LIN {X 0,Y 301.473,Z 710.898,A -85,B 0,C 180,E1 14594.697,E2 14594.697} C_VEL
LIN {X 0,Y 299.686,Z 720.643,A -85,B 0,C 180,E1 14592.72,E2 14592.72} C_VEL
LIN {X 0,Y 297.823,Z 729.269,A -85,B 0,C 180,E1 14590.444,E2 14590.444} C_VEL
LIN {X 0,Y 296.157,Z 735.724,A -85,B 0,C 180,E1 14588.151,E2 14588.151} C_VEL
LIN {X 0,Y 294.632,Z 740.781,A -85,B 0,C 180,E1 14585.647,E2 14585.647} C_VEL
LIN {X 0,Y 293.317,Z 744.193,A -85,B 0,C 180,E1 14582.93,E2 14582.93} C_VEL
LIN {X 0,Y 292.262,Z 745.687,A -85,B 0,C 180,E1 14579.999,E2 14579.999} C_VEL
LIN {X 0,Y 291.583,Z 745.107,A -85,B 0,C 180,E1 14577.168,E2 14577.168} C_VEL
LIN {X 0,Y 291.215,Z 742.755,A -85,B 0,C 180,E1 14574.483,E2 14574.483} C_VEL
LIN {X 0,Y 291.115,Z 738.842,A -85,B 0,C 180,E1 14571.904,E2 14571.904} C_VEL
LIN {X 0,Y 291.269,Z 732.598,A -85,B 0,C 180,E1 14569.116,E2 14569.116} C_VEL
LIN {X 0,Y 291.687,Z 724.621,A -85,B 0,C 180,E1 14566.52,E2 14566.52} C_VEL
LIN {X 0,Y 292.312,Z 714.997,A -85,B 0,C 180,E1 14564.118,E2 14564.118} C_VEL
LIN {X 0,Y 293.088,Z 703.694,A -85,B 0,C 180,E1 14561.913,E2 14561.913} C_VEL
LIN {X 0,Y 293.954,Z 690.528,A -85,B 0,C 180,E1 14559.906,E2 14559.906} C_VEL
LIN {X 0,Y 294.781,Z 675.92,A -85,B 0,C 180,E1 14558.197,E2 14558.197} C_VEL
LIN {X 0,Y 295.446,Z 660.979,A -85,B 0,C 180,E1 14556.885,E2 14556.885} C_VEL
LIN {X 0,Y 295.895,Z 644.769,A -85,B 0,C 180,E1 14555.878,E2 14555.878} C_VEL
LIN {X 0,Y 296.067,Z 626.386,A -85,B 0,C 180,E1 14555.173,E2 14555.173} C_VEL
LIN {X 0,Y 297.336,Z 577.945,A -85,B 0,C 180,E1 14553.621,E2 14553.621} C_VEL
LIN {X 0,Y 298.083,Z 578.111,A -85,B 0,C 180,E1 14553.289,E2 14553.289} C_VEL
LIN {X 0,Y 299.719,Z 576.086,A -85,B 0,C 180,E1 14552.857,E2 14552.857} C_VEL
LIN {X 0,Y 302.62,Z 570.153,A -85,B 0,C 180,E1 14552.375,E2 14552.375} C_VEL
LIN {X 0,Y 306.801,Z 558.743,A -85,B 0,C 180,E1 14551.96,E2 14551.96} C_VEL
LIN {X 0,Y 307.694,Z 556.167,A -85,B 0,C 180,E1 14551.888,E2 14551.888} C_VEL
LIN {X 0,Y 310.325,Z 552.374,A -85,B 0,C 180,E1 14551.283,E2 14551.283} C_VEL
LIN {X 0,Y 313.629,Z 545.368,A -85,B 0,C 180,E1 14550.753,E2 14550.753} C_VEL
LIN {X 0,Y 317.925,Z 533.318,A -85,B 0,C 180,E1 14550.308,E2 14550.308} C_VEL
LIN {X 0,Y 319.018,Z 529.98,A -85,B 0,C 180,E1 14550.213,E2 14550.213} C_VEL
LIN {X 0,Y 323.323,Z 523.899,A -85,B 0,C 180,E1 14549.272,E2 14549.272} C_VEL
LIN {X 0,Y 329.072,Z 514.334,A -85,B 0,C 180,E1 14548.185,E2 14548.185} C_VEL
LIN {X 0,Y 333.692,Z 509.138,A -85,B 0,C 180,E1 14547.182,E2 14547.182} C_VEL
LIN {X 0,Y 338.897,Z 501.157,A -85,B 0,C 180,E1 14546.236,E2 14546.236} C_VEL
LIN {X 0,Y 340.375,Z 498.972,A -85,B 0,C 180,E1 14545.971,E2 14545.971} C_VEL
LIN {X 0,Y 345.61,Z 492.984,A -85,B 0,C 180,E1 14544.958,E2 14544.958} C_VEL
LIN {X 0,Y 351.852,Z 483.792,A -85,B 0,C 180,E1 14543.917,E2 14543.917} C_VEL
LIN {X 0,Y 356.859,Z 478.438,A -85,B 0,C 180,E1 14543.023,E2 14543.023} C_VEL
LIN {X 0,Y 350.683,Z 533.515,A -85,B 0,C 180,E1 14541.496,E2 14541.496} C_VEL
LIN {X 0,Y 343.595,Z 587.069,A -85,B 0,C 180,E1 14539.73,E2 14539.73} C_VEL
LIN {X 0,Y 340.274,Z 612.573,A -85,B 0,C 180,E1 14538.644,E2 14538.644} C_VEL
LIN {X 0,Y 336.94,Z 632.228,A -85,B 0,C 180,E1 14537.512,E2 14537.512} C_VEL
LIN {X 0,Y 332.931,Z 651.111,A -85,B 0,C 180,E1 14536.119,E2 14536.119} C_VEL
LIN {X 0,Y 328.102,Z 670.254,A -85,B 0,C 180,E1 14534.334,E2 14534.334} C_VEL
LIN {X 0,Y 322.92,Z 688.102,A -85,B 0,C 180,E1 14532.266,E2 14532.266} C_VEL
LIN {X 0,Y 317.65,Z 704.404,A -85,B 0,C 180,E1 14529.951,E2 14529.951} C_VEL
LIN {X 0,Y 312.389,Z 719.507,A -85,B 0,C 180,E1 14527.339,E2 14527.339} C_VEL
LIN {X 0,Y 307.364,Z 733.168,A -85,B 0,C 180,E1 14524.474,E2 14524.474} C_VEL
LIN {X 0,Y 302.603,Z 745.779,A -85,B 0,C 180,E1 14521.249,E2 14521.249} C_VEL
LIN {X 0,Y 298.41,Z 756.887,A -85,B 0,C 180,E1 14517.758,E2 14517.758} C_VEL
LIN {X 0,Y 294.914,Z 766.473,A -85,B 0,C 180,E1 14514.007,E2 14514.007} C_VEL
LIN {X 0,Y 292.324,Z 774.116,A -85,B 0,C 180,E1 14510.21,E2 14510.21} C_VEL
LIN {X 0,Y 290.465,Z 780.308,A -85,B 0,C 180,E1 14506.176,E2 14506.176} C_VEL
LIN {X 0,Y 289.38,Z 784.674,A -85,B 0,C 180,E1 14502.167,E2 14502.167} C_VEL
LIN {X 0,Y 288.847,Z 787.269,A -85,B 0,C 180,E1 14498.36,E2 14498.36} C_VEL
LIN {X 0,Y 288.632,Z 788.437,A -85,B 0,C 180,E1 14494.371,E2 14494.371} C_VEL
LIN {X 0,Y 288.641,Z 788.017,A -85,B 0,C 180,E1 14490.397,E2 14490.397} C_VEL
LIN {X 0,Y 288.874,Z 786.163,A -85,B 0,C 180,E1 14486.627,E2 14486.627} C_VEL
LIN {X 0,Y 289.451,Z 782.871,A -85,B 0,C 180,E1 14482.856,E2 14482.856} C_VEL
LIN {X 0,Y 290.598,Z 777.745,A -85,B 0,C 180,E1 14478.891,E2 14478.891} C_VEL
LIN {X 0,Y 291.846,Z 772.956,A -85,B 0,C 180,E1 14476.075,E2 14476.075} C_VEL
LIN {X 0,Y 291.661,Z 770.405,A -85,B 0,C 180,E1 14474.638,E2 14474.638} C_VEL
LIN {X 0,Y 288.214,Z 763.219,A -85,B 0,C 180,E1 14470.745,E2 14470.745} C_VEL
LIN {X 0,Y 288.512,Z 760.327,A -85,B 0,C 180,E1 14469.546,E2 14469.546} C_VEL
LIN {X 0,Y 292.227,Z 749.899,A -85,B 0,C 180,E1 14465.973,E2 14465.973} C_VEL
LIN {X 0,Y 296.474,Z 738.2,A -85,B 0,C 180,E1 14462.699,E2 14462.699} C_VEL
LIN {X 0,Y 301.185,Z 725.063,A -85,B 0,C 180,E1 14459.672,E2 14459.672} C_VEL
LIN {X 0,Y 306.278,Z 710.292,A -85,B 0,C 180,E1 14456.871,E2 14456.871} C_VEL
LIN {X 0,Y 311.276,Z 694.805,A -85,B 0,C 180,E1 14454.451,E2 14454.451} C_VEL
LIN {X 0,Y 316.243,Z 677.951,A -85,B 0,C 180,E1 14452.281,E2 14452.281} C_VEL
LIN {X 0,Y 320.912,Z 660.2,A -85,B 0,C 180,E1 14450.42,E2 14450.42} C_VEL
LIN {X 0,Y 324.977,Z 642.253,A -85,B 0,C 180,E1 14448.897,E2 14448.897} C_VEL
LIN {X 0,Y 328.596,Z 622.858,A -85,B 0,C 180,E1 14447.59,E2 14447.59} C_VEL
LIN {X 0,Y 331.499,Z 602.817,A -85,B 0,C 180,E1 14446.562,E2 14446.562} C_VEL
LIN {X 0,Y 336.631,Z 562.875,A -85,B 0,C 180,E1 14445.046,E2 14445.046} C_VEL
LIN {X 0,Y 343.508,Z 506.974,A -85,B 0,C 180,E1 14443.314,E2 14443.314} C_VEL
LIN {X 0,Y 348.719,Z 454.242,A -85,B 0,C 180,E1 14441.938,E2 14441.938} C_VEL
LIN {X 0,Y 352.555,Z 400.926,A -85,B 0,C 180,E1 14440.775,E2 14440.775} C_VEL
LIN {X 0,Y 352.938,Z 393.306,A -85,B 0,C 180,E1 14440.603,E2 14440.603} C_VEL
LIN {X 0,Y 344.835,Z 382.448,A -85,B 0,C 180,E1 14438.327,E2 14438.327} C_VEL
LIN {X 0,Y 335.306,Z 391.656,A -85,B 0,C 180,E1 14436.188,E2 14436.188} C_VEL
LIN {X 0,Y 329.497,Z 398.011,A -85,B 0,C 180,E1 14434.785,E2 14434.785} C_VEL
LIN {X 0,Y 325.165,Z 402.639,A -85,B 0,C 180,E1 14433.66,E2 14433.66} C_VEL
LIN {X 0,Y 319.752,Z 409.849,A -85,B 0,C 180,E1 14432.219,E2 14432.219} C_VEL
LIN {X 0,Y 314.779,Z 421.202,A -85,B 0,C 180,E1 14431.023,E2 14431.023} C_VEL
LIN {X 0,Y 311.088,Z 427.898,A -85,B 0,C 180,E1 14429.987,E2 14429.987} C_VEL
LIN {X 0,Y 308.623,Z 431.225,A -85,B 0,C 180,E1 14429.196,E2 14429.196} C_VEL
LIN {X 0,Y 303.63,Z 444,A -85,B 0,C 180,E1 14427.853,E2 14427.853} C_VEL
LIN {X 0,Y 300.278,Z 450.967,A -85,B 0,C 180,E1 14426.794,E2 14426.794} C_VEL
LIN {X 0,Y 298.518,Z 453.454,A -85,B 0,C 180,E1 14426.133,E2 14426.133} C_VEL
LIN {X 0,Y 297.997,Z 453.855,A -85,B 0,C 180,E1 14425.888,E2 14425.888} C_VEL
LIN {X 0,Y 296.772,Z 468.599,A -85,B 0,C 180,E1 14424.405,E2 14424.405} C_VEL
LIN {X 0,Y 296.008,Z 473.564,A -85,B 0,C 180,E1 14424.006,E2 14424.006} C_VEL
LIN {X 0,Y 290.441,Z 604.08,A -85,B 0,C 180,E1 14419.652,E2 14419.652} C_VEL
LIN {X 0,Y 290.011,Z 625.296,A -85,B 0,C 180,E1 14418.793,E2 14418.793} C_VEL
LIN {X 0,Y 289.326,Z 642.963,A -85,B 0,C 180,E1 14417.706,E2 14417.706} C_VEL
LIN {X 0,Y 288.352,Z 660.558,A -85,B 0,C 180,E1 14416.209,E2 14416.209} C_VEL
LIN {X 0,Y 287.212,Z 677.45,A -85,B 0,C 180,E1 14414.311,E2 14414.311} C_VEL
LIN {X 0,Y 286.035,Z 692.745,A -85,B 0,C 180,E1 14412.108,E2 14412.108} C_VEL
LIN {X 0,Y 284.951,Z 706.521,A -85,B 0,C 180,E1 14409.598,E2 14409.598} C_VEL
LIN {X 0,Y 284.135,Z 717.555,A -85,B 0,C 180,E1 14407.075,E2 14407.075} C_VEL
LIN {X 0,Y 283.579,Z 726.784,A -85,B 0,C 180,E1 14404.45,E2 14404.45} C_VEL
LIN {X 0,Y 283.252,Z 735.102,A -85,B 0,C 180,E1 14401.417,E2 14401.417} C_VEL
LIN {X 0,Y 283.252,Z 741.235,A -85,B 0,C 180,E1 14398.383,E2 14398.383} C_VEL
LIN {X 0,Y 283.544,Z 745.254,A -85,B 0,C 180,E1 14395.551,E2 14395.551} C_VEL
LIN {X 0,Y 284.166,Z 747.725,A -85,B 0,C 180,E1 14392.52,E2 14392.52} C_VEL
LIN {X 0,Y 285.075,Z 748.436,A -85,B 0,C 180,E1 14389.696,E2 14389.696} C_VEL
LIN {X 0,Y 286.424,Z 747.35,A -85,B 0,C 180,E1 14386.68,E2 14386.68} C_VEL
LIN {X 0,Y 288.052,Z 744.664,A -85,B 0,C 180,E1 14383.878,E2 14383.878} C_VEL
LIN {X 0,Y 290.06,Z 740.16,A -85,B 0,C 180,E1 14381.094,E2 14381.094} C_VEL
LIN {X 0,Y 292.467,Z 733.68,A -85,B 0,C 180,E1 14378.333,E2 14378.333} C_VEL
LIN {X 0,Y 295.04,Z 725.576,A -85,B 0,C 180,E1 14375.792,E2 14375.792} C_VEL
LIN {X 0,Y 297.684,Z 715.934,A -85,B 0,C 180,E1 14373.467,E2 14373.467} C_VEL
LIN {X 0,Y 300.337,Z 704.849,A -85,B 0,C 180,E1 14371.355,E2 14371.355} C_VEL
LIN {X 0,Y 303.037,Z 691.567,A -85,B 0,C 180,E1 14369.352,E2 14369.352} C_VEL
LIN {X 0,Y 305.593,Z 676.279,A -85,B 0,C 180,E1 14367.549,E2 14367.549} C_VEL
LIN {X 0,Y 307.814,Z 659.516,A -85,B 0,C 180,E1 14366.035,E2 14366.035} C_VEL
LIN {X 0,Y 309.452,Z 643.901,A -85,B 0,C 180,E1 14364.949,E2 14364.949} C_VEL
LIN {X 0,Y 312.209,Z 641.947,A -85,B 0,C 180,E1 14364.574,E2 14364.574} C_VEL
LIN {X 0,Y 315.963,Z 637.407,A -85,B 0,C 180,E1 14364.279,E2 14364.279} C_VEL
LIN {X 0,Y 318.626,Z 632.886,A -85,B 0,C 180,E1 14364.181,E2 14364.181} C_VEL
LIN {X 0,Y 322.084,Z 629.461,A -85,B 0,C 180,E1 14363.817,E2 14363.817} C_VEL
LIN {X 0,Y 326.321,Z 623.421,A -85,B 0,C 180,E1 14363.529,E2 14363.529} C_VEL
LIN {X 0,Y 329.749,Z 617.515,A -85,B 0,C 180,E1 14363.375,E2 14363.375} C_VEL
LIN {X 0,Y 334.495,Z 611.357,A -85,B 0,C 180,E1 14362.965,E2 14362.965} C_VEL
LIN {X 0,Y 339.904,Z 601.538,A -85,B 0,C 180,E1 14362.673,E2 14362.673} C_VEL
LIN {X 0,Y 341.058,Z 599.168,A -85,B 0,C 180,E1 14362.623,E2 14362.623} C_VEL
LIN {X 0,Y 336.007,Z 627.852,A -85,B 0,C 180,E1 14361.432,E2 14361.432} C_VEL
LIN {X 0,Y 330.753,Z 653.868,A -85,B 0,C 180,E1 14360.025,E2 14360.025} C_VEL
LIN {X 0,Y 325.14,Z 679.325,A -85,B 0,C 180,E1 14358.27,E2 14358.27} C_VEL
LIN {X 0,Y 319.358,Z 703.464,A -85,B 0,C 180,E1 14356.219,E2 14356.219} C_VEL
LIN {X 0,Y 314.203,Z 722.714,A -85,B 0,C 180,E1 14354.179,E2 14354.179} C_VEL
LIN {X 0,Y 309.087,Z 739.953,A -85,B 0,C 180,E1 14351.926,E2 14351.926} C_VEL
LIN {X 0,Y 303.589,Z 756.816,A -85,B 0,C 180,E1 14349.224,E2 14349.224} C_VEL
LIN {X 0,Y 298.58,Z 771.612,A -85,B 0,C 180,E1 14346.351,E2 14346.351} C_VEL
LIN {X 0,Y 293.647,Z 785.695,A -85,B 0,C 180,E1 14343.011,E2 14343.011} C_VEL
LIN {X 0,Y 289.342,Z 798.276,A -85,B 0,C 180,E1 14339.387,E2 14339.387} C_VEL
LIN {X 0,Y 285.795,Z 809.244,A -85,B 0,C 180,E1 14335.488,E2 14335.488} C_VEL
LIN {X 0,Y 283.125,Z 818.695,A -85,B 0,C 180,E1 14331.33,E2 14331.33} C_VEL
LIN {X 0,Y 281.424,Z 826.219,A -85,B 0,C 180,E1 14327.117,E2 14327.117} C_VEL
LIN {X 0,Y 280.547,Z 832.143,A -85,B 0,C 180,E1 14322.766,E2 14322.766} C_VEL
LIN {X 0,Y 280.318,Z 836.176,A -85,B 0,C 180,E1 14318.616,E2 14318.616} C_VEL
LIN {X 0,Y 280.394,Z 838.536,A -85,B 0,C 180,E1 14314.704,E2 14314.704} C_VEL
LIN {X 0,Y 280.478,Z 839.547,A -85,B 0,C 180,E1 14310.817,E2 14310.817} C_VEL
LIN {X 0,Y 280.429,Z 839.233,A -85,B 0,C 180,E1 14306.934,E2 14306.934} C_VEL
LIN {X 0,Y 280.319,Z 837.595,A -85,B 0,C 180,E1 14303.034,E2 14303.034} C_VEL
LIN {X 0,Y 280.377,Z 834.425,A -85,B 0,C 180,E1 14298.897,E2 14298.897} C_VEL
LIN {X 0,Y 280.979,Z 829.386,A -85,B 0,C 180,E1 14294.521,E2 14294.521} C_VEL
LIN {X 0,Y 282.433,Z 822.567,A -85,B 0,C 180,E1 14290.132,E2 14290.132} C_VEL
LIN {X 0,Y 284.789,Z 814.229,A -85,B 0,C 180,E1 14285.967,E2 14285.967} C_VEL
LIN {X 0,Y 288.424,Z 803.331,A -85,B 0,C 180,E1 14281.645,E2 14281.645} C_VEL
LIN {X 0,Y 292.672,Z 791.63,A -85,B 0,C 180,E1 14277.912,E2 14277.912} C_VEL
LIN {X 0,Y 297.922,Z 777.604,A -85,B 0,C 180,E1 14274.27,E2 14274.27} C_VEL
LIN {X 0,Y 303.283,Z 763.18,A -85,B 0,C 180,E1 14271.215,E2 14271.215} C_VEL
LIN {X 0,Y 309.187,Z 746.554,A -85,B 0,C 180,E1 14268.332,E2 14268.332} C_VEL
LIN {X 0,Y 314.815,Z 729.546,A -85,B 0,C 180,E1 14265.928,E2 14265.928} C_VEL
LIN {X 0,Y 320.081,Z 711.951,A -85,B 0,C 180,E1 14263.905,E2 14263.905} C_VEL
LIN {X 0,Y 324.783,Z 694.187,A -85,B 0,C 180,E1 14262.235,E2 14262.235} C_VEL
LIN {X 0,Y 330.423,Z 671.409,A -85,B 0,C 180,E1 14260.444,E2 14260.444} C_VEL
LIN {X 0,Y 336.265,Z 645.855,A -85,B 0,C 180,E1 14258.827,E2 14258.827} C_VEL
LIN {X 0,Y 341.881,Z 618.451,A -85,B 0,C 180,E1 14257.485,E2 14257.485} C_VEL
LIN {X 0,Y 346.787,Z 589.883,A -85,B 0,C 180,E1 14256.411,E2 14256.411} C_VEL
LIN {X 0,Y 349.983,Z 567.917,A -85,B 0,C 180,E1 14255.797,E2 14255.797} C_VEL
LIN {X 0,Y 353.901,Z 543.241,A -85,B 0,C 180,E1 14255.513,E2 14255.513} C_VEL
LIN {X 0,Y 355.166,Z 534.693,A -85,B 0,C 180,E1 14255.47,E2 14255.47} C_VEL
LIN {X 0,Y 346.998,Z 514.246,A -85,B 0,C 180,E1 14252.898,E2 14252.898} C_VEL
LIN {X 0,Y 342.19,Z 498.864,A -85,B 0,C 180,E1 14251.115,E2 14251.115} C_VEL
LIN {X 0,Y 338.758,Z 503.075,A -85,B 0,C 180,E1 14250.361,E2 14250.361} C_VEL
LIN {X 0,Y 333.41,Z 513.045,A -85,B 0,C 180,E1 14249.262,E2 14249.262} C_VEL
LIN {X 0,Y 331.124,Z 516.93,A -85,B 0,C 180,E1 14248.754,E2 14248.754} C_VEL
LIN {X 0,Y 325.481,Z 529.287,A -85,B 0,C 180,E1 14247.611,E2 14247.611} C_VEL
LIN {X 0,Y 318.157,Z 545.033,A -85,B 0,C 180,E1 14246.189,E2 14246.189} C_VEL
LIN {X 0,Y 311.572,Z 565.14,A -85,B 0,C 180,E1 14245.506,E2 14245.506} C_VEL
LIN {X 0,Y 307.707,Z 574.04,A -85,B 0,C 180,E1 14244.962,E2 14244.962} C_VEL
LIN {X 0,Y 306.249,Z 576.987,A -85,B 0,C 180,E1 14244.676,E2 14244.676} C_VEL
LIN {X 0,Y 301.442,Z 633.673,A -85,B 0,C 180,E1 14242.435,E2 14242.435} C_VEL
LIN {X 0,Y 300.381,Z 660.053,A -85,B 0,C 180,E1 14241.196,E2 14241.196} C_VEL
LIN {X 0,Y 299.511,Z 674.161,A -85,B 0,C 180,E1 14240.213,E2 14240.213} C_VEL
LIN {X 0,Y 298.152,Z 688.209,A -85,B 0,C 180,E1 14238.881,E2 14238.881} C_VEL
LIN {X 0,Y 296.484,Z 701.18,A -85,B 0,C 180,E1 14237.263,E2 14237.263} C_VEL
LIN {X 0,Y 294.653,Z 712.217,A -85,B 0,C 180,E1 14235.481,E2 14235.481} C_VEL
LIN {X 0,Y 292.688,Z 722.167,A -85,B 0,C 180,E1 14233.432,E2 14233.432} C_VEL
LIN {X 0,Y 290.642,Z 730.739,A -85,B 0,C 180,E1 14231.107,E2 14231.107} C_VEL
LIN {X 0,Y 288.692,Z 737.689,A -85,B 0,C 180,E1 14228.564,E2 14228.564} C_VEL
LIN {X 0,Y 287.034,Z 742.578,A -85,B 0,C 180,E1 14225.998,E2 14225.998} C_VEL
LIN {X 0,Y 285.603,Z 745.838,A -85,B 0,C 180,E1 14223.21,E2 14223.21} C_VEL
LIN {X 0,Y 284.522,Z 747.18,A -85,B 0,C 180,E1 14220.402,E2 14220.402} C_VEL
LIN {X 0,Y 283.767,Z 746.63,A -85,B 0,C 180,E1 14217.576,E2 14217.576} C_VEL
LIN {X 0,Y 283.351,Z 744.475,A -85,B 0,C 180,E1 14214.938,E2 14214.938} C_VEL
LIN {X 0,Y 283.185,Z 740.308,A -85,B 0,C 180,E1 14212.084,E2 14212.084} C_VEL
LIN {X 0,Y 283.317,Z 734.044,A -85,B 0,C 180,E1 14209.219,E2 14209.219} C_VEL
LIN {X 0,Y 283.727,Z 726.067,A -85,B 0,C 180,E1 14206.55,E2 14206.55} C_VEL
LIN {X 0,Y 284.358,Z 716.452,A -85,B 0,C 180,E1 14204.081,E2 14204.081} C_VEL
LIN {X 0,Y 285.149,Z 705.131,A -85,B 0,C 180,E1 14201.815,E2 14201.815} C_VEL
LIN {X 0,Y 286.038,Z 691.955,A -85,B 0,C 180,E1 14199.753,E2 14199.753} C_VEL
LIN {X 0,Y 286.902,Z 677.151,A -85,B 0,C 180,E1 14197.976,E2 14197.976} C_VEL
LIN {X 0,Y 287.597,Z 661.945,A -85,B 0,C 180,E1 14196.611,E2 14196.611} C_VEL
LIN {X 0,Y 288.063,Z 645.959,A -85,B 0,C 180,E1 14195.595,E2 14195.595} C_VEL
LIN {X 0,Y 288.255,Z 627.249,A -85,B 0,C 180,E1 14194.854,E2 14194.854} C_VEL
LIN {X 0,Y 288.75,Z 603.42,A -85,B 0,C 180,E1 14194.021,E2 14194.021} C_VEL
LIN {X 0,Y 289.539,Z 603.619,A -85,B 0,C 180,E1 14193.656,E2 14193.656} C_VEL
LIN {X 0,Y 291.248,Z 601.636,A -85,B 0,C 180,E1 14193.201,E2 14193.201} C_VEL
LIN {X 0,Y 294.153,Z 596.042,A -85,B 0,C 180,E1 14192.725,E2 14192.725} C_VEL
LIN {X 0,Y 298.315,Z 585.446,A -85,B 0,C 180,E1 14192.34,E2 14192.34} C_VEL
LIN {X 0,Y 298.798,Z 584.326,A -85,B 0,C 180,E1 14192.28,E2 14192.28} C_VEL
LIN {X 0,Y 301.447,Z 580.726,A -85,B 0,C 180,E1 14191.658,E2 14191.658} C_VEL
LIN {X 0,Y 304.858,Z 574.047,A -85,B 0,C 180,E1 14191.116,E2 14191.116} C_VEL
LIN {X 0,Y 309.255,Z 562.611,A -85,B 0,C 180,E1 14190.682,E2 14190.682} C_VEL
LIN {X 0,Y 310.163,Z 560.384,A -85,B 0,C 180,E1 14190.579,E2 14190.579} C_VEL
LIN {X 0,Y 313.547,Z 554.777,A -85,B 0,C 180,E1 14189.93,E2 14189.93} C_VEL
LIN {X 0,Y 317.447,Z 546.013,A -85,B 0,C 180,E1 14189.398,E2 14189.398} C_VEL
LIN {X 0,Y 321.678,Z 534.312,A -85,B 0,C 180,E1 14188.989,E2 14188.989} C_VEL
LIN {X 0,Y 327.825,Z 525.172,A -85,B 0,C 180,E1 14187.792,E2 14187.792} C_VEL
LIN {X 0,Y 330.859,Z 520.239,A -85,B 0,C 180,E1 14187.252,E2 14187.252} C_VEL
LIN {X 0,Y 336.05,Z 514.248,A -85,B 0,C 180,E1 14186.193,E2 14186.193} C_VEL
LIN {X 0,Y 341.775,Z 505.555,A -85,B 0,C 180,E1 14185.216,E2 14185.216} C_VEL
LIN {X 0,Y 348.007,Z 498.402,A -85,B 0,C 180,E1 14184.067,E2 14184.067} C_VEL
LIN {X 0,Y 350.504,Z 495.083,A -85,B 0,C 180,E1 14183.652,E2 14183.652} C_VEL
LIN {X 0,Y 343.831,Z 549.112,A -85,B 0,C 180,E1 14182.074,E2 14182.074} C_VEL
LIN {X 0,Y 337.573,Z 594.457,A -85,B 0,C 180,E1 14180.488,E2 14180.488} C_VEL
LIN {X 0,Y 334.298,Z 617.469,A -85,B 0,C 180,E1 14179.438,E2 14179.438} C_VEL
LIN {X 0,Y 330.58,Z 637.491,A -85,B 0,C 180,E1 14178.207,E2 14178.207} C_VEL
LIN {X 0,Y 326.131,Z 656.786,A -85,B 0,C 180,E1 14176.685,E2 14176.685} C_VEL
LIN {X 0,Y 321.332,Z 674.476,A -85,B 0,C 180,E1 14174.938,E2 14174.938} C_VEL
LIN {X 0,Y 316.045,Z 691.625,A -85,B 0,C 180,E1 14172.859,E2 14172.859} C_VEL
LIN {X 0,Y 310.315,Z 708.386,A -85,B 0,C 180,E1 14170.364,E2 14170.364} C_VEL
LIN {X 0,Y 304.734,Z 723.436,A -85,B 0,C 180,E1 14167.61,E2 14167.61} C_VEL
LIN {X 0,Y 299.447,Z 736.974,A -85,B 0,C 180,E1 14164.586,E2 14164.586} C_VEL
LIN {X 0,Y 294.434,Z 749.487,A -85,B 0,C 180,E1 14161.155,E2 14161.155} C_VEL
LIN {X 0,Y 290.14,Z 760.241,A -85,B 0,C 180,E1 14157.502,E2 14157.502} C_VEL
LIN {X 0,Y 286.662,Z 769.297,A -85,B 0,C 180,E1 14153.648,E2 14153.648} C_VEL
LIN {X 0,Y 284.112,Z 776.483,A -85,B 0,C 180,E1 14149.746,E2 14149.746} C_VEL
LIN {X 0,Y 282.318,Z 782.213,A -85,B 0,C 180,E1 14145.615,E2 14145.615} C_VEL
LIN {X 0,Y 281.299,Z 786.19,A -85,B 0,C 180,E1 14141.481,E2 14141.481} C_VEL
LIN {X 0,Y 280.83,Z 788.452,A -85,B 0,C 180,E1 14137.57,E2 14137.57} C_VEL
LIN {X 0,Y 280.655,Z 789.247,A -85,B 0,C 180,E1 14133.472,E2 14133.472} C_VEL
LIN {X 0,Y 280.715,Z 788.494,A -85,B 0,C 180,E1 14129.592,E2 14129.592} C_VEL
LIN {X 0,Y 281.014,Z 786.329,A -85,B 0,C 180,E1 14125.715,E2 14125.715} C_VEL
LIN {X 0,Y 281.775,Z 782.486,A -85,B 0,C 180,E1 14121.635,E2 14121.635} C_VEL
LIN {X 0,Y 283.171,Z 776.95,A -85,B 0,C 180,E1 14117.562,E2 14117.562} C_VEL
LIN {X 0,Y 285.395,Z 769.595,A -85,B 0,C 180,E1 14113.514,E2 14113.514} C_VEL
LIN {X 0,Y 288.361,Z 760.758,A -85,B 0,C 180,E1 14109.712,E2 14109.712} C_VEL
LIN {X 0,Y 288.512,Z 760.327,A -85,B 0,C 180,E1 14109.546,E2 14109.546} C_VEL
LIN {X 0,Y 288.845,Z 756.908,A -85,B 0,C 180,E1 14108.166,E2 14108.166} C_VEL
LIN {X 0,Y 286.851,Z 748.129,A -85,B 0,C 180,E1 14104.586,E2 14104.586} C_VEL
LIN {X 0,Y 287.58,Z 743.998,A -85,B 0,C 180,E1 14103.272,E2 14103.272} C_VEL
LIN {X 0,Y 292.4,Z 731.332,A -85,B 0,C 180,E1 14100.05,E2 14100.05} C_VEL
LIN {X 0,Y 297.715,Z 716.915,A -85,B 0,C 180,E1 14097.039,E2 14097.039} C_VEL
LIN {X 0,Y 303.299,Z 700.848,A -85,B 0,C 180,E1 14094.303,E2 14094.303} C_VEL
LIN {X 0,Y 308.555,Z 684.249,A -85,B 0,C 180,E1 14091.998,E2 14091.998} C_VEL
LIN {X 0,Y 313.53,Z 666.737,A -85,B 0,C 180,E1 14090.014,E2 14090.014} C_VEL
LIN {X 0,Y 318.143,Z 647.977,A -85,B 0,C 180,E1 14088.302,E2 14088.302} C_VEL
LIN {X 0,Y 322.06,Z 628.877,A -85,B 0,C 180,E1 14086.921,E2 14086.921} C_VEL
LIN {X 0,Y 325.211,Z 609.441,A -85,B 0,C 180,E1 14085.832,E2 14085.832} C_VEL
LIN {X 0,Y 329.868,Z 574.362,A -85,B 0,C 180,E1 14084.399,E2 14084.399} C_VEL
LIN {X 0,Y 337.033,Z 520.261,A -85,B 0,C 180,E1 14082.638,E2 14082.638} C_VEL
LIN {X 0,Y 342.733,Z 467.47,A -85,B 0,C 180,E1 14081.194,E2 14081.194} C_VEL
LIN {X 0,Y 346.898,Z 416.197,A -85,B 0,C 180,E1 14080.026,E2 14080.026} C_VEL
LIN {X 0,Y 348.024,Z 397.545,A -85,B 0,C 180,E1 14079.629,E2 14079.629} C_VEL
LIN {X 0,Y 343.595,Z 391.743,A -85,B 0,C 180,E1 14078.358,E2 14078.358} C_VEL
LIN {X 0,Y 336.308,Z 399.076,A -85,B 0,C 180,E1 14076.751,E2 14076.751} C_VEL
LIN {X 0,Y 330.857,Z 404.904,A -85,B 0,C 180,E1 14075.467,E2 14075.467} C_VEL
LIN {X 0,Y 325.093,Z 411.229,A -85,B 0,C 180,E1 14074.014,E2 14074.014} C_VEL
LIN {X 0,Y 321.814,Z 415.767,A -85,B 0,C 180,E1 14073.177,E2 14073.177} C_VEL
LIN {X 0,Y 316.612,Z 427.101,A -85,B 0,C 180,E1 14071.963,E2 14071.963} C_VEL
LIN {X 0,Y 312.483,Z 434.231,A -85,B 0,C 180,E1 14070.848,E2 14070.848} C_VEL
LIN {X 0,Y 310.32,Z 437.349,A -85,B 0,C 180,E1 14070.202,E2 14070.202} C_VEL
LIN {X 0,Y 305.021,Z 450.105,A -85,B 0,C 180,E1 14068.835,E2 14068.835} C_VEL
LIN {X 0,Y 301.378,Z 457.188,A -85,B 0,C 180,E1 14067.73,E2 14067.73} C_VEL
LIN {X 0,Y 299.019,Z 460.764,A -85,B 0,C 180,E1 14066.902,E2 14066.902} C_VEL
LIN {X 0,Y 293.641,Z 475.605,A -85,B 0,C 180,E1 14065.448,E2 14065.448} C_VEL
LIN {X 0,Y 290.016,Z 488.364,A -85,B 0,C 180,E1 14064.711,E2 14064.711} C_VEL
LIN {X 0,Y 288.155,Z 493.193,A -85,B 0,C 180,E1 14064.171,E2 14064.171} C_VEL
LIN {X 0,Y 287.441,Z 494.48,A -85,B 0,C 180,E1 14063.86,E2 14063.86} C_VEL
LIN {X 0,Y 282.665,Z 604.848,A -85,B 0,C 180,E1 14060.014,E2 14060.014} C_VEL
LIN {X 0,Y 282.2,Z 626.495,A -85,B 0,C 180,E1 14059.112,E2 14059.112} C_VEL
LIN {X 0,Y 281.492,Z 644.075,A -85,B 0,C 180,E1 14058.001,E2 14058.001} C_VEL
LIN {X 0,Y 280.503,Z 661.451,A -85,B 0,C 180,E1 14056.491,E2 14056.491} C_VEL
LIN {X 0,Y 279.367,Z 677.882,A -85,B 0,C 180,E1 14054.616,E2 14054.616} C_VEL
LIN {X 0,Y 278.247,Z 692.07,A -85,B 0,C 180,E1 14052.557,E2 14052.557} C_VEL
LIN {X 0,Y 277.222,Z 704.752,A -85,B 0,C 180,E1 14050.285,E2 14050.285} C_VEL
LIN {X 0,Y 276.333,Z 716.457,A -85,B 0,C 180,E1 14047.695,E2 14047.695} C_VEL
LIN {X 0,Y 275.671,Z 726.876,A -85,B 0,C 180,E1 14044.786,E2 14044.786} C_VEL
LIN {X 0,Y 275.331,Z 735.054,A -85,B 0,C 180,E1 14041.874,E2 14041.874} C_VEL
LIN {X 0,Y 275.303,Z 741.687,A -85,B 0,C 180,E1 14038.752,E2 14038.752} C_VEL
LIN {X 0,Y 275.65,Z 746.567,A -85,B 0,C 180,E1 14035.424,E2 14035.424} C_VEL
LIN {X 0,Y 276.337,Z 749.212,A -85,B 0,C 180,E1 14032.307,E2 14032.307} C_VEL
LIN {X 0,Y 277.424,Z 750.081,A -85,B 0,C 180,E1 14029.199,E2 14029.199} C_VEL
LIN {X 0,Y 278.922,Z 749.03,A -85,B 0,C 180,E1 14026.104,E2 14026.104} C_VEL
LIN {X 0,Y 280.733,Z 746.415,A -85,B 0,C 180,E1 14023.233,E2 14023.233} C_VEL
LIN {X 0,Y 283.122,Z 741.563,A -85,B 0,C 180,E1 14020.183,E2 14020.183} C_VEL
LIN {X 0,Y 285.606,Z 735.511,A -85,B 0,C 180,E1 14017.552,E2 14017.552} C_VEL
LIN {X 0,Y 288.404,Z 727.547,A -85,B 0,C 180,E1 14014.979,E2 14014.979} C_VEL
LIN {X 0,Y 291.297,Z 718.064,A -85,B 0,C 180,E1 14012.617,E2 14012.617} C_VEL
LIN {X 0,Y 294.244,Z 707.059,A -85,B 0,C 180,E1 14010.448,E2 14010.448} C_VEL
LIN {X 0,Y 297.309,Z 693.608,A -85,B 0,C 180,E1 14008.357,E2 14008.357} C_VEL
LIN {X 0,Y 300.13,Z 678.694,A -85,B 0,C 180,E1 14006.541,E2 14006.541} C_VEL
LIN {X 0,Y 302.578,Z 662.738,A -85,B 0,C 180,E1 14005.036,E2 14005.036} C_VEL
LIN {X 0,Y 303.267,Z 657.999,A -85,B 0,C 180,E1 14004.647,E2 14004.647} C_VEL
LIN {X 0,Y 306.275,Z 656.194,A -85,B 0,C 180,E1 14004.243,E2 14004.243} C_VEL
LIN {X 0,Y 309.957,Z 652.257,A -85,B 0,C 180,E1 14003.935,E2 14003.935} C_VEL
LIN {X 0,Y 312.119,Z 649.255,A -85,B 0,C 180,E1 14003.831,E2 14003.831} C_VEL
LIN {X 0,Y 316.297,Z 645.47,A -85,B 0,C 180,E1 14003.411,E2 14003.411} C_VEL
LIN {X 0,Y 320.875,Z 639.296,A -85,B 0,C 180,E1 14003.142,E2 14003.142} C_VEL
LIN {X 0,Y 322.154,Z 637.336,A -85,B 0,C 180,E1 14003.091,E2 14003.091} C_VEL
LIN {X 0,Y 326.855,Z 632.084,A -85,B 0,C 180,E1 14002.689,E2 14002.689} C_VEL
LIN {X 0,Y 330.624,Z 626.5,A -85,B 0,C 180,E1 14002.481,E2 14002.481} C_VEL
LIN {X 0,Y 325.202,Z 652.699,A -85,B 0,C 180,E1 14001.066,E2 14001.066} C_VEL
LIN {X 0,Y 319.17,Z 679.283,A -85,B 0,C 180,E1 13999.229,E2 13999.229} C_VEL
LIN {X 0,Y 313.157,Z 703.459,A -85,B 0,C 180,E1 13997.151,E2 13997.151} C_VEL
LIN {X 0,Y 307.796,Z 722.673,A -85,B 0,C 180,E1 13995.086,E2 13995.086} C_VEL
LIN {X 0,Y 302.427,Z 739.918,A -85,B 0,C 180,E1 13992.782,E2 13992.782} C_VEL
LIN {X 0,Y 296.751,Z 756.625,A -85,B 0,C 180,E1 13990.057,E2 13990.057} C_VEL
LIN {X 0,Y 291.514,Z 771.316,A -85,B 0,C 180,E1 13987.133,E2 13987.133} C_VEL
LIN {X 0,Y 286.357,Z 785.361,A -85,B 0,C 180,E1 13983.723,E2 13983.723} C_VEL
LIN {X 0,Y 281.843,Z 797.896,A -85,B 0,C 180,E1 13980.014,E2 13980.014} C_VEL
LIN {X 0,Y 277.943,Z 809.34,A -85,B 0,C 180,E1 13975.803,E2 13975.803} C_VEL
LIN {X 0,Y 275.183,Z 818.64,A -85,B 0,C 180,E1 13971.529,E2 13971.529} C_VEL
LIN {X 0,Y 273.382,Z 826.298,A -85,B 0,C 180,E1 13967.013,E2 13967.013} C_VEL
LIN {X 0,Y 272.538,Z 831.954,A -85,B 0,C 180,E1 13962.614,E2 13962.614} C_VEL
LIN {X 0,Y 272.343,Z 835.86,A -85,B 0,C 180,E1 13958.232,E2 13958.232} C_VEL
LIN {X 0,Y 272.436,Z 838.043,A -85,B 0,C 180,E1 13954.209,E2 13954.209} C_VEL
LIN {X 0,Y 272.515,Z 838.872,A -85,B 0,C 180,E1 13950.21,E2 13950.21} C_VEL
LIN {X 0,Y 272.432,Z 838.365,A -85,B 0,C 180,E1 13946.212,E2 13946.212} C_VEL
LIN {X 0,Y 272.323,Z 836.525,A -85,B 0,C 180,E1 13942.192,E2 13942.192} C_VEL
LIN {X 0,Y 272.46,Z 833.082,A -85,B 0,C 180,E1 13937.926,E2 13937.926} C_VEL
LIN {X 0,Y 273.25,Z 827.791,A -85,B 0,C 180,E1 13933.416,E2 13933.416} C_VEL
LIN {X 0,Y 274.972,Z 820.697,A -85,B 0,C 180,E1 13928.9,E2 13928.9} C_VEL
LIN {X 0,Y 277.841,Z 811.555,A -85,B 0,C 180,E1 13924.415,E2 13924.415} C_VEL
LIN {X 0,Y 281.531,Z 801.392,A -85,B 0,C 180,E1 13920.418,E2 13920.418} C_VEL
LIN {X 0,Y 286.3,Z 789.042,A -85,B 0,C 180,E1 13916.51,E2 13916.51} C_VEL
LIN {X 0,Y 291.689,Z 775.475,A -85,B 0,C 180,E1 13913.004,E2 13913.004} C_VEL
LIN {X 0,Y 297.361,Z 760.789,A -85,B 0,C 180,E1 13909.916,E2 13909.916} C_VEL
LIN {X 0,Y 303.32,Z 744.747,A -85,B 0,C 180,E1 13907.147,E2 13907.147} C_VEL
LIN {X 0,Y 309.117,Z 727.872,A -85,B 0,C 180,E1 13904.766,E2 13904.766} C_VEL
LIN {X 0,Y 314.8,Z 709.501,A -85,B 0,C 180,E1 13902.668,E2 13902.668} C_VEL
LIN {X 0,Y 320.058,Z 690.177,A -85,B 0,C 180,E1 13900.886,E2 13900.886} C_VEL
LIN {X 0,Y 326.231,Z 665.644,A -85,B 0,C 180,E1 13899.036,E2 13899.036} C_VEL
LIN {X 0,Y 332.388,Z 638.845,A -85,B 0,C 180,E1 13897.425,E2 13897.425} C_VEL
LIN {X 0,Y 338.137,Z 610.893,A -85,B 0,C 180,E1 13896.147,E2 13896.147} C_VEL
LIN {X 0,Y 343.219,Z 580.059,A -85,B 0,C 180,E1 13895.054,E2 13895.054} C_VEL
LIN {X 0,Y 346.437,Z 559.693,A -85,B 0,C 180,E1 13894.617,E2 13894.617} C_VEL
LIN {X 0,Y 349.938,Z 537.417,A -85,B 0,C 180,E1 13894.428,E2 13894.428} C_VEL
LIN {X 0,Y 342.577,Z 517.901,A -85,B 0,C 180,E1 13891.937,E2 13891.937} C_VEL
LIN {X 0,Y 340.204,Z 510.75,A -85,B 0,C 180,E1 13891.05,E2 13891.05} C_VEL
LIN {X 0,Y 334.85,Z 520.05,A -85,B 0,C 180,E1 13889.96,E2 13889.96} C_VEL
LIN {X 0,Y 333.264,Z 523.16,A -85,B 0,C 180,E1 13889.647,E2 13889.647} C_VEL
LIN {X 0,Y 327.358,Z 535.331,A -85,B 0,C 180,E1 13888.505,E2 13888.505} C_VEL
LIN {X 0,Y 320.768,Z 549.42,A -85,B 0,C 180,E1 13887.33,E2 13887.33} C_VEL
LIN {X 0,Y 315.352,Z 566.098,A -85,B 0,C 180,E1 13886.834,E2 13886.834} C_VEL
LIN {X 0,Y 310.723,Z 576.895,A -85,B 0,C 180,E1 13886.26,E2 13886.26} C_VEL
LIN {X 0,Y 308.716,Z 580.825,A -85,B 0,C 180,E1 13885.964,E2 13885.964} C_VEL
LIN {X 0,Y 303.588,Z 593.844,A -85,B 0,C 180,E1 13885.546,E2 13885.546} C_VEL
LIN {X 0,Y 299.711,Z 601.292,A -85,B 0,C 180,E1 13885.04,E2 13885.04} C_VEL
LIN {X 0,Y 298.254,Z 603.855,A -85,B 0,C 180,E1 13884.76,E2 13884.76} C_VEL
LIN {X 0,Y 295.067,Z 643.386,A -85,B 0,C 180,E1 13883.073,E2 13883.073} C_VEL
LIN {X 0,Y 294.154,Z 663.595,A -85,B 0,C 180,E1 13882.021,E2 13882.021} C_VEL
LIN {X 0,Y 293.007,Z 678.517,A -85,B 0,C 180,E1 13880.891,E2 13880.891} C_VEL
LIN {X 0,Y 291.519,Z 691.847,A -85,B 0,C 180,E1 13879.536,E2 13879.536} C_VEL
LIN {X 0,Y 289.673,Z 704.196,A -85,B 0,C 180,E1 13877.89,E2 13877.89} C_VEL
LIN {X 0,Y 287.667,Z 715.108,A -85,B 0,C 180,E1 13876.04,E2 13876.04} C_VEL
LIN {X 0,Y 285.566,Z 724.576,A -85,B 0,C 180,E1 13873.98,E2 13873.98} C_VEL
LIN {X 0,Y 283.369,Z 732.965,A -85,B 0,C 180,E1 13871.602,E2 13871.602} C_VEL
LIN {X 0,Y 281.254,Z 739.698,A -85,B 0,C 180,E1 13868.998,E2 13868.998} C_VEL
LIN {X 0,Y 279.457,Z 744.41,A -85,B 0,C 180,E1 13866.367,E2 13866.367} C_VEL
LIN {X 0,Y 278.003,Z 747.37,A -85,B 0,C 180,E1 13863.711,E2 13863.711} C_VEL
LIN {X 0,Y 276.797,Z 748.677,A -85,B 0,C 180,E1 13860.827,E2 13860.827} C_VEL
LIN {X 0,Y 275.949,Z 748.116,A -85,B 0,C 180,E1 13857.923,E2 13857.923} C_VEL
LIN {X 0,Y 275.467,Z 745.943,A -85,B 0,C 180,E1 13855.21,E2 13855.21} C_VEL
LIN {X 0,Y 275.257,Z 741.764,A -85,B 0,C 180,E1 13852.275,E2 13852.275} C_VEL
LIN {X 0,Y 275.363,Z 735.475,A -85,B 0,C 180,E1 13849.327,E2 13849.327} C_VEL
LIN {X 0,Y 275.76,Z 727.453,A -85,B 0,C 180,E1 13846.581,E2 13846.581} C_VEL
LIN {X 0,Y 276.395,Z 717.789,A -85,B 0,C 180,E1 13844.041,E2 13844.041} C_VEL
LIN {X 0,Y 277.204,Z 706.462,A -85,B 0,C 180,E1 13841.711,E2 13841.711} C_VEL
LIN {X 0,Y 278.12,Z 693.297,A -85,B 0,C 180,E1 13839.59,E2 13839.59} C_VEL
LIN {X 0,Y 279.009,Z 678.64,A -85,B 0,C 180,E1 13837.773,E2 13837.773} C_VEL
LIN {X 0,Y 279.743,Z 663.222,A -85,B 0,C 180,E1 13836.346,E2 13836.346} C_VEL
LIN {X 0,Y 280.237,Z 647.18,A -85,B 0,C 180,E1 13835.298,E2 13835.298} C_VEL
LIN {X 0,Y 280.442,Z 628.642,A -85,B 0,C 180,E1 13834.539,E2 13834.539} C_VEL
LIN {X 0,Y 280.505,Z 625.823,A -85,B 0,C 180,E1 13834.413,E2 13834.413} C_VEL
LIN {X 0,Y 281.175,Z 626.12,A -85,B 0,C 180,E1 13834.062,E2 13834.062} C_VEL
LIN {X 0,Y 282.257,Z 625.31,A -85,B 0,C 180,E1 13833.717,E2 13833.717} C_VEL
LIN {X 0,Y 284.459,Z 622.113,A -85,B 0,C 180,E1 13833.261,E2 13833.261} C_VEL
LIN {X 0,Y 288.017,Z 614.601,A -85,B 0,C 180,E1 13832.823,E2 13832.823} C_VEL
LIN {X 0,Y 289.967,Z 609.958,A -85,B 0,C 180,E1 13832.646,E2 13832.646} C_VEL
LIN {X 0,Y 292.732,Z 606.496,A -85,B 0,C 180,E1 13831.988,E2 13831.988} C_VEL
LIN {X 0,Y 296.156,Z 600.209,A -85,B 0,C 180,E1 13831.44,E2 13831.44} C_VEL
LIN {X 0,Y 300.532,Z 589.625,A -85,B 0,C 180,E1 13831.023,E2 13831.023} C_VEL
LIN {X 0,Y 301.986,Z 587.429,A -85,B 0,C 180,E1 13830.739,E2 13830.739} C_VEL
LIN {X 0,Y 305.598,Z 581.32,A -85,B 0,C 180,E1 13830.101,E2 13830.101} C_VEL
LIN {X 0,Y 309.787,Z 571.921,A -85,B 0,C 180,E1 13829.601,E2 13829.601} C_VEL
LIN {X 0,Y 312.658,Z 564.488,A -85,B 0,C 180,E1 13829.345,E2 13829.345} C_VEL
LIN {X 0,Y 316.675,Z 557.525,A -85,B 0,C 180,E1 13828.655,E2 13828.655} C_VEL
LIN {X 0,Y 321.061,Z 547.578,A -85,B 0,C 180,E1 13828.125,E2 13828.125} C_VEL
LIN {X 0,Y 324.452,Z 538.542,A -85,B 0,C 180,E1 13827.808,E2 13827.808} C_VEL
LIN {X 0,Y 332.113,Z 526.868,A -85,B 0,C 180,E1 13826.438,E2 13826.438} C_VEL
LIN {X 0,Y 338.866,Z 518.862,A -85,B 0,C 180,E1 13825.158,E2 13825.158} C_VEL
LIN {X 0,Y 344.103,Z 511.177,A -85,B 0,C 180,E1 13824.299,E2 13824.299} C_VEL
LIN {X 0,Y 337.008,Z 563.704,A -85,B 0,C 180,E1 13822.685,E2 13822.685} C_VEL
LIN {X 0,Y 331.401,Z 602.831,A -85,B 0,C 180,E1 13821.219,E2 13821.219} C_VEL
LIN {X 0,Y 328.109,Z 623.797,A -85,B 0,C 180,E1 13820.169,E2 13820.169} C_VEL
LIN {X 0,Y 324.022,Z 643.673,A -85,B 0,C 180,E1 13818.845,E2 13818.845} C_VEL
LIN {X 0,Y 319.293,Z 662.469,A -85,B 0,C 180,E1 13817.253,E2 13817.253} C_VEL
LIN {X 0,Y 314.005,Z 680.415,A -85,B 0,C 180,E1 13815.357,E2 13815.357} C_VEL
LIN {X 0,Y 308.215,Z 697.802,A -85,B 0,C 180,E1 13813.082,E2 13813.082} C_VEL
LIN {X 0,Y 302.173,Z 714.23,A -85,B 0,C 180,E1 13810.432,E2 13810.432} C_VEL
LIN {X 0,Y 296.439,Z 728.711,A -85,B 0,C 180,E1 13807.567,E2 13807.567} C_VEL
LIN {X 0,Y 290.89,Z 742.107,A -85,B 0,C 180,E1 13804.313,E2 13804.313} C_VEL
LIN {X 0,Y 285.811,Z 754.101,A -85,B 0,C 180,E1 13800.715,E2 13800.715} C_VEL
LIN {X 0,Y 281.459,Z 764.497,A -85,B 0,C 180,E1 13796.818,E2 13796.818} C_VEL
LIN {X 0,Y 277.952,Z 773.226,A -85,B 0,C 180,E1 13792.638,E2 13792.638} C_VEL
LIN {X 0,Y 275.483,Z 779.974,A -85,B 0,C 180,E1 13788.407,E2 13788.407} C_VEL
LIN {X 0,Y 273.937,Z 784.912,A -85,B 0,C 180,E1 13784.155,E2 13784.155} C_VEL
LIN {X 0,Y 273.103,Z 788.151,A -85,B 0,C 180,E1 13779.908,E2 13779.908} C_VEL
LIN {X 0,Y 272.747,Z 789.76,A -85,B 0,C 180,E1 13775.681,E2 13775.681} C_VEL
LIN {X 0,Y 272.683,Z 789.78,A -85,B 0,C 180,E1 13771.681,E2 13771.681} C_VEL
LIN {X 0,Y 272.855,Z 788.386,A -85,B 0,C 180,E1 13767.69,E2 13767.69} C_VEL
LIN {X 0,Y 273.404,Z 785.385,A -85,B 0,C 180,E1 13763.49,E2 13763.49} C_VEL
LIN {X 0,Y 274.528,Z 780.737,A -85,B 0,C 180,E1 13759.295,E2 13759.295} C_VEL
LIN {X 0,Y 276.443,Z 774.337,A -85,B 0,C 180,E1 13755.12,E2 13755.12} C_VEL
LIN {X 0,Y 279.272,Z 766.05,A -85,B 0,C 180,E1 13750.986,E2 13750.986} C_VEL
LIN {X 0,Y 282.898,Z 756.229,A -85,B 0,C 180,E1 13747.121,E2 13747.121} C_VEL
LIN {X 0,Y 287.217,Z 744.92,A -85,B 0,C 180,E1 13743.539,E2 13743.539} C_VEL
LIN {X 0,Y 287.58,Z 743.998,A -85,B 0,C 180,E1 13743.272,E2 13743.272} C_VEL
LIN {X 0,Y 288.419,Z 739.809,A -85,B 0,C 180,E1 13741.981,E2 13741.981} C_VEL
LIN {X 0,Y 287.689,Z 729.061,A -85,B 0,C 180,E1 13738.597,E2 13738.597} C_VEL
LIN {X 0,Y 288.738,Z 724.137,A -85,B 0,C 180,E1 13737.423,E2 13737.423} C_VEL
LIN {X 0,Y 294.204,Z 709.55,A -85,B 0,C 180,E1 13734.653,E2 13734.653} C_VEL
LIN {X 0,Y 299.789,Z 693.424,A -85,B 0,C 180,E1 13732.144,E2 13732.144} C_VEL
LIN {X 0,Y 305.024,Z 676.761,A -85,B 0,C 180,E1 13730.023,E2 13730.023} C_VEL
LIN {X 0,Y 309.98,Z 658.858,A -85,B 0,C 180,E1 13728.169,E2 13728.169} C_VEL
LIN {X 0,Y 314.406,Z 640.091,A -85,B 0,C 180,E1 13726.613,E2 13726.613} C_VEL
LIN {X 0,Y 318.071,Z 620.993,A -85,B 0,C 180,E1 13725.366,E2 13725.366} C_VEL
LIN {X 0,Y 321.191,Z 600.053,A -85,B 0,C 180,E1 13724.332,E2 13724.332} C_VEL
LIN {X 0,Y 327.19,Z 557.637,A -85,B 0,C 180,E1 13722.728,E2 13722.728} C_VEL
LIN {X 0,Y 334.079,Z 504.443,A -85,B 0,C 180,E1 13721.084,E2 13721.084} C_VEL
LIN {X 0,Y 339.378,Z 453.367,A -85,B 0,C 180,E1 13719.757,E2 13719.757} C_VEL
LIN {X 0,Y 343.234,Z 401.981,A -85,B 0,C 180,E1 13718.64,E2 13718.64} C_VEL
LIN {X 0,Y 342.54,Z 401.308,A -85,B 0,C 180,E1 13718.444,E2 13718.444} C_VEL
LIN {X 0,Y 337.955,Z 405.766,A -85,B 0,C 180,E1 13717.445,E2 13717.445} C_VEL
LIN {X 0,Y 331.963,Z 412.122,A -85,B 0,C 180,E1 13716.075,E2 13716.075} C_VEL
LIN {X 0,Y 326.679,Z 417.792,A -85,B 0,C 180,E1 13714.781,E2 13714.781} C_VEL
LIN {X 0,Y 323.967,Z 421.633,A -85,B 0,C 180,E1 13714.121,E2 13714.121} C_VEL
LIN {X 0,Y 318.501,Z 432.976,A -85,B 0,C 180,E1 13712.895,E2 13712.895} C_VEL
LIN {X 0,Y 314.067,Z 440.364,A -85,B 0,C 180,E1 13711.742,E2 13711.742} C_VEL
LIN {X 0,Y 312.205,Z 443.126,A -85,B 0,C 180,E1 13711.223,E2 13711.223} C_VEL
LIN {X 0,Y 306.576,Z 455.955,A -85,B 0,C 180,E1 13709.837,E2 13709.837} C_VEL
LIN {X 0,Y 302.508,Z 463.394,A -85,B 0,C 180,E1 13708.665,E2 13708.665} C_VEL
LIN {X 0,Y 300.417,Z 466.675,A -85,B 0,C 180,E1 13707.989,E2 13707.989} C_VEL
LIN {X 0,Y 295.796,Z 478.856,A -85,B 0,C 180,E1 13706.819,E2 13706.819} C_VEL
LIN {X 0,Y 291.949,Z 491.785,A -85,B 0,C 180,E1 13706.083,E2 13706.083} C_VEL
LIN {X 0,Y 289.552,Z 497.904,A -85,B 0,C 180,E1 13705.436,E2 13705.436} C_VEL
LIN {X 0,Y 288.94,Z 499.487,A -85,B 0,C 180,E1 13705.267,E2 13705.267} C_VEL
LIN {X 0,Y 284.219,Z 517.151,A -85,B 0,C 180,E1 13704.652,E2 13704.652} C_VEL
LIN {X 0,Y 280.712,Z 527.957,A -85,B 0,C 180,E1 13703.972,E2 13703.972} C_VEL
LIN {X 0,Y 278.683,Z 532.72,A -85,B 0,C 180,E1 13703.385,E2 13703.385} C_VEL
LIN {X 0,Y 277.855,Z 534.032,A -85,B 0,C 180,E1 13702.997,E2 13702.997} C_VEL
LIN {X 0,Y 274.849,Z 608.06,A -85,B 0,C 180,E1 13700.302,E2 13700.302} C_VEL
LIN {X 0,Y 274.384,Z 627.955,A -85,B 0,C 180,E1 13699.429,E2 13699.429} C_VEL
LIN {X 0,Y 273.622,Z 645.744,A -85,B 0,C 180,E1 13698.256,E2 13698.256} C_VEL
LIN {X 0,Y 272.614,Z 662.671,A -85,B 0,C 180,E1 13696.734,E2 13696.734} C_VEL
LIN {X 0,Y 271.394,Z 679.681,A -85,B 0,C 180,E1 13694.727,E2 13694.727} C_VEL
LIN {X 0,Y 270.154,Z 695.104,A -85,B 0,C 180,E1 13692.397,E2 13692.397} C_VEL
LIN {X 0,Y 269.055,Z 708.518,A -85,B 0,C 180,E1 13689.844,E2 13689.844} C_VEL
LIN {X 0,Y 268.237,Z 719.387,A -85,B 0,C 180,E1 13687.282,E2 13687.282} C_VEL
LIN {X 0,Y 267.663,Z 728.912,A -85,B 0,C 180,E1 13684.5,E2 13684.5} C_VEL
LIN {X 0,Y 267.354,Z 736.955,A -85,B 0,C 180,E1 13681.501,E2 13681.501} C_VEL
LIN {X 0,Y 267.378,Z 743.164,A -85,B 0,C 180,E1 13678.501,E2 13678.501} C_VEL
LIN {X 0,Y 267.795,Z 748.11,A -85,B 0,C 180,E1 13675.074,E2 13675.074} C_VEL
LIN {X 0,Y 268.576,Z 750.807,A -85,B 0,C 180,E1 13671.868,E2 13671.868} C_VEL
LIN {X 0,Y 269.796,Z 751.735,A -85,B 0,C 180,E1 13668.673,E2 13668.673} C_VEL
LIN {X 0,Y 271.463,Z 750.76,A -85,B 0,C 180,E1 13665.496,E2 13665.496} C_VEL
LIN {X 0,Y 273.624,Z 747.941,A -85,B 0,C 180,E1 13662.345,E2 13662.345} C_VEL
LIN {X 0,Y 276.296,Z 743.053,A -85,B 0,C 180,E1 13659.229,E2 13659.229} C_VEL
LIN {X 0,Y 279.064,Z 736.88,A -85,B 0,C 180,E1 13656.524,E2 13656.524} C_VEL
LIN {X 0,Y 282.141,Z 729.01,A -85,B 0,C 180,E1 13653.933,E2 13653.933} C_VEL
LIN {X 0,Y 285.612,Z 718.681,A -85,B 0,C 180,E1 13651.341,E2 13651.341} C_VEL
LIN {X 0,Y 289.118,Z 706.546,A -85,B 0,C 180,E1 13648.984,E2 13648.984} C_VEL
LIN {X 0,Y 292.411,Z 693.227,A -85,B 0,C 180,E1 13646.95,E2 13646.95} C_VEL
LIN {X 0,Y 295.397,Z 679.004,A -85,B 0,C 180,E1 13645.227,E2 13645.227} C_VEL
LIN {X 0,Y 297.023,Z 670.818,A -85,B 0,C 180,E1 13644.384,E2 13644.384} C_VEL
LIN {X 0,Y 300.481,Z 668.743,A -85,B 0,C 180,E1 13643.917,E2 13643.917} C_VEL
LIN {X 0,Y 304.305,Z 665.028,A -85,B 0,C 180,E1 13643.611,E2 13643.611} C_VEL
LIN {X 0,Y 305.826,Z 663.462,A -85,B 0,C 180,E1 13643.486,E2 13643.486} C_VEL
LIN {X 0,Y 310.382,Z 659.696,A -85,B 0,C 180,E1 13643.026,E2 13643.026} C_VEL
LIN {X 0,Y 315.512,Z 653.756,A -85,B 0,C 180,E1 13642.695,E2 13642.695} C_VEL
LIN {X 0,Y 320.358,Z 648.952,A -85,B 0,C 180,E1 13642.302,E2 13642.302} C_VEL
LIN {X 0,Y 314.181,Z 675.435,A -85,B 0,C 180,E1 13640.511,E2 13640.511} C_VEL
LIN {X 0,Y 308.221,Z 699.129,A -85,B 0,C 180,E1 13638.535,E2 13638.535} C_VEL
LIN {X 0,Y 302.87,Z 718,A -85,B 0,C 180,E1 13636.576,E2 13636.576} C_VEL
LIN {X 0,Y 297.182,Z 735.946,A -85,B 0,C 180,E1 13634.264,E2 13634.264} C_VEL
LIN {X 0,Y 291.233,Z 752.979,A -85,B 0,C 180,E1 13631.546,E2 13631.546} C_VEL
LIN {X 0,Y 285.37,Z 768.771,A -85,B 0,C 180,E1 13628.456,E2 13628.456} C_VEL
LIN {X 0,Y 280.006,Z 782.743,A -85,B 0,C 180,E1 13625.093,E2 13625.093} C_VEL
LIN {X 0,Y 275.094,Z 795.576,A -85,B 0,C 180,E1 13621.316,E2 13621.316} C_VEL
LIN {X 0,Y 271.186,Z 806.282,A -85,B 0,C 180,E1 13617.444,E2 13617.444} C_VEL
LIN {X 0,Y 267.859,Z 816.469,A -85,B 0,C 180,E1 13612.843,E2 13612.843} C_VEL
LIN {X 0,Y 265.817,Z 824.154,A -85,B 0,C 180,E1 13608.419,E2 13608.419} C_VEL
LIN {X 0,Y 264.69,Z 830.292,A -85,B 0,C 180,E1 13603.767,E2 13603.767} C_VEL
LIN {X 0,Y 264.366,Z 834.485,A -85,B 0,C 180,E1 13599.36,E2 13599.36} C_VEL
LIN {X 0,Y 264.432,Z 836.981,A -85,B 0,C 180,E1 13595.207,E2 13595.207} C_VEL
LIN {X 0,Y 264.539,Z 838.095,A -85,B 0,C 180,E1 13591.083,E2 13591.083} C_VEL
LIN {X 0,Y 264.495,Z 837.914,A -85,B 0,C 180,E1 13587.183,E2 13587.183} C_VEL
LIN {X 0,Y 264.363,Z 836.408,A -85,B 0,C 180,E1 13583.048,E2 13583.048} C_VEL
LIN {X 0,Y 264.414,Z 833.357,A -85,B 0,C 180,E1 13578.66,E2 13578.66} C_VEL
LIN {X 0,Y 265.084,Z 828.511,A -85,B 0,C 180,E1 13574.017,E2 13574.017} C_VEL
LIN {X 0,Y 266.707,Z 821.802,A -85,B 0,C 180,E1 13569.366,E2 13569.366} C_VEL
LIN {X 0,Y 269.498,Z 813.184,A -85,B 0,C 180,E1 13564.744,E2 13564.744} C_VEL
LIN {X 0,Y 273.366,Z 802.882,A -85,B 0,C 180,E1 13560.411,E2 13560.411} C_VEL
LIN {X 0,Y 278.196,Z 791.044,A -85,B 0,C 180,E1 13556.393,E2 13556.393} C_VEL
LIN {X 0,Y 283.611,Z 778.012,A -85,B 0,C 180,E1 13552.82,E2 13552.82} C_VEL
LIN {X 0,Y 289.835,Z 762.867,A -85,B 0,C 180,E1 13549.437,E2 13549.437} C_VEL
LIN {X 0,Y 295.806,Z 747.688,A -85,B 0,C 180,E1 13546.672,E2 13546.672} C_VEL
LIN {X 0,Y 302.133,Z 730.317,A -85,B 0,C 180,E1 13544.099,E2 13544.099} C_VEL
LIN {X 0,Y 308.021,Z 712.547,A -85,B 0,C 180,E1 13541.965,E2 13541.965} C_VEL
LIN {X 0,Y 313.656,Z 692.98,A -85,B 0,C 180,E1 13540.084,E2 13540.084} C_VEL
LIN {X 0,Y 320.29,Z 667.654,A -85,B 0,C 180,E1 13538.123,E2 13538.123} C_VEL
LIN {X 0,Y 326.554,Z 641.474,A -85,B 0,C 180,E1 13536.511,E2 13536.511} C_VEL
LIN {X 0,Y 332.853,Z 612.053,A -85,B 0,C 180,E1 13535.133,E2 13535.133} C_VEL
LIN {X 0,Y 338.118,Z 581.518,A -85,B 0,C 180,E1 13534.03,E2 13534.03} C_VEL
LIN {X 0,Y 341.466,Z 560.862,A -85,B 0,C 180,E1 13533.563,E2 13533.563} C_VEL
LIN {X 0,Y 344.808,Z 539.963,A -85,B 0,C 180,E1 13533.342,E2 13533.342} C_VEL
LIN {X 0,Y 338.737,Z 523.346,A -85,B 0,C 180,E1 13531.15,E2 13531.15} C_VEL
LIN {X 0,Y 336.363,Z 527.339,A -85,B 0,C 180,E1 13530.687,E2 13530.687} C_VEL
LIN {X 0,Y 330.13,Z 539.85,A -85,B 0,C 180,E1 13529.554,E2 13529.554} C_VEL
LIN {X 0,Y 323.998,Z 552.606,A -85,B 0,C 180,E1 13528.525,E2 13528.525} C_VEL
LIN {X 0,Y 318.363,Z 569.427,A -85,B 0,C 180,E1 13528.037,E2 13528.037} C_VEL
LIN {X 0,Y 313.425,Z 580.621,A -85,B 0,C 180,E1 13527.462,E2 13527.462} C_VEL
LIN {X 0,Y 311.573,Z 584.335,A -85,B 0,C 180,E1 13527.219,E2 13527.219} C_VEL
LIN {X 0,Y 306.097,Z 597.649,A -85,B 0,C 180,E1 13526.793,E2 13526.793} C_VEL
LIN {X 0,Y 301.757,Z 605.686,A -85,B 0,C 180,E1 13526.253,E2 13526.253} C_VEL
LIN {X 0,Y 300.423,Z 608.028,A -85,B 0,C 180,E1 13526.085,E2 13526.085} C_VEL
LIN {X 0,Y 295.802,Z 618.012,A -85,B 0,C 180,E1 13525.743,E2 13525.743} C_VEL
LIN {X 0,Y 292.388,Z 623.682,A -85,B 0,C 180,E1 13525.305,E2 13525.305} C_VEL
LIN {X 0,Y 290.81,Z 626.007,A -85,B 0,C 180,E1 13525.003,E2 13525.003} C_VEL
LIN {X 0,Y 288.604,Z 658.746,A -85,B 0,C 180,E1 13523.426,E2 13523.426} C_VEL
LIN {X 0,Y 287.542,Z 674.197,A -85,B 0,C 180,E1 13522.38,E2 13522.38} C_VEL
LIN {X 0,Y 286.035,Z 687.965,A -85,B 0,C 180,E1 13521.102,E2 13521.102} C_VEL
LIN {X 0,Y 284.012,Z 701.505,A -85,B 0,C 180,E1 13519.431,E2 13519.431} C_VEL
LIN {X 0,Y 281.915,Z 712.739,A -85,B 0,C 180,E1 13517.652,E2 13517.652} C_VEL
LIN {X 0,Y 279.561,Z 722.987,A -85,B 0,C 180,E1 13515.559,E2 13515.559} C_VEL
LIN {X 0,Y 277.089,Z 732.124,A -85,B 0,C 180,E1 13513.139,E2 13513.139} C_VEL
LIN {X 0,Y 274.682,Z 739.482,A -85,B 0,C 180,E1 13510.486,E2 13510.486} C_VEL
LIN {X 0,Y 272.611,Z 744.763,A -85,B 0,C 180,E1 13507.799,E2 13507.799} C_VEL
LIN {X 0,Y 270.888,Z 748.189,A -85,B 0,C 180,E1 13505.081,E2 13505.081} C_VEL
LIN {X 0,Y 269.435,Z 750.031,A -85,B 0,C 180,E1 13502.126,E2 13502.126} C_VEL
LIN {X 0,Y 268.378,Z 749.972,A -85,B 0,C 180,E1 13499.145,E2 13499.145} C_VEL
LIN {X 0,Y 267.687,Z 748.048,A -85,B 0,C 180,E1 13496.144,E2 13496.144} C_VEL
LIN {X 0,Y 267.367,Z 744.587,A -85,B 0,C 180,E1 13493.342,E2 13493.342} C_VEL
LIN {X 0,Y 267.347,Z 738.888,A -85,B 0,C 180,E1 13490.31,E2 13490.31} C_VEL
LIN {X 0,Y 267.64,Z 731.537,A -85,B 0,C 180,E1 13487.485,E2 13487.485} C_VEL
LIN {X 0,Y 268.188,Z 722.635,A -85,B 0,C 180,E1 13484.871,E2 13484.871} C_VEL
LIN {X 0,Y 268.974,Z 711.666,A -85,B 0,C 180,E1 13482.364,E2 13482.364} C_VEL
LIN {X 0,Y 269.895,Z 698.844,A -85,B 0,C 180,E1 13480.072,E2 13480.072} C_VEL
LIN {X 0,Y 270.831,Z 684.617,A -85,B 0,C 180,E1 13478.106,E2 13478.106} C_VEL
LIN {X 0,Y 271.645,Z 669.401,A -85,B 0,C 180,E1 13476.513,E2 13476.513} C_VEL
LIN {X 0,Y 272.265,Z 653.532,A -85,B 0,C 180,E1 13475.308,E2 13475.308} C_VEL
LIN {X 0,Y 272.515,Z 644.284,A -85,B 0,C 180,E1 13474.752,E2 13474.752} C_VEL
LIN {X 0,Y 273.602,Z 644.319,A -85,B 0,C 180,E1 13474.222,E2 13474.222} C_VEL
LIN {X 0,Y 275.511,Z 642.495,A -85,B 0,C 180,E1 13473.72,E2 13473.72} C_VEL
LIN {X 0,Y 278.103,Z 638.596,A -85,B 0,C 180,E1 13473.293,E2 13473.293} C_VEL
LIN {X 0,Y 281.286,Z 632.537,A -85,B 0,C 180,E1 13472.992,E2 13472.992} C_VEL
LIN {X 0,Y 284.076,Z 629.526,A -85,B 0,C 180,E1 13472.315,E2 13472.315} C_VEL
LIN {X 0,Y 287.434,Z 624.102,A -85,B 0,C 180,E1 13471.764,E2 13471.764} C_VEL
LIN {X 0,Y 291.581,Z 615.118,A -85,B 0,C 180,E1 13471.359,E2 13471.359} C_VEL
LIN {X 0,Y 295.571,Z 609.389,A -85,B 0,C 180,E1 13470.57,E2 13470.57} C_VEL
LIN {X 0,Y 299.602,Z 601.654,A -85,B 0,C 180,E1 13470.029,E2 13470.029} C_VEL
LIN {X 0,Y 303.34,Z 592.974,A -85,B 0,C 180,E1 13469.677,E2 13469.677} C_VEL
LIN {X 0,Y 307.446,Z 586.386,A -85,B 0,C 180,E1 13468.971,E2 13468.971} C_VEL
LIN {X 0,Y 311.89,Z 577.035,A -85,B 0,C 180,E1 13468.43,E2 13468.43} C_VEL
LIN {X 0,Y 315.426,Z 568.302,A -85,B 0,C 180,E1 13468.117,E2 13468.117} C_VEL
LIN {X 0,Y 320.009,Z 560.206,A -85,B 0,C 180,E1 13467.412,E2 13467.412} C_VEL
LIN {X 0,Y 324.843,Z 549.099,A -85,B 0,C 180,E1 13466.883,E2 13466.883} C_VEL
LIN {X 0,Y 327.283,Z 542.768,A -85,B 0,C 180,E1 13466.665,E2 13466.665} C_VEL
LIN {X 0,Y 334.833,Z 531.694,A -85,B 0,C 180,E1 13465.38,E2 13465.38} C_VEL
LIN {X 0,Y 337.351,Z 529.033,A -85,B 0,C 180,E1 13464.9,E2 13464.9} C_VEL
LIN {X 0,Y 329.56,Z 582.102,A -85,B 0,C 180,E1 13463.159,E2 13463.159} C_VEL
LIN {X 0,Y 324.773,Z 614.278,A -85,B 0,C 180,E1 13461.795,E2 13461.795} C_VEL
LIN {X 0,Y 321.18,Z 633.549,A -85,B 0,C 180,E1 13460.679,E2 13460.679} C_VEL
LIN {X 0,Y 316.712,Z 652.625,A -85,B 0,C 180,E1 13459.261,E2 13459.261} C_VEL
LIN {X 0,Y 311.38,Z 671.589,A -85,B 0,C 180,E1 13457.472,E2 13457.472} C_VEL
LIN {X 0,Y 305.598,Z 689.351,A -85,B 0,C 180,E1 13455.381,E2 13455.381} C_VEL
LIN {X 0,Y 299.461,Z 706.167,A -85,B 0,C 180,E1 13452.932,E2 13452.932} C_VEL
LIN {X 0,Y 293.214,Z 721.787,A -85,B 0,C 180,E1 13450.128,E2 13450.128} C_VEL
LIN {X 0,Y 287.24,Z 735.81,A -85,B 0,C 180,E1 13447.028,E2 13447.028} C_VEL
LIN {X 0,Y 281.697,Z 748.33,A -85,B 0,C 180,E1 13443.622,E2 13443.622} C_VEL
LIN {X 0,Y 276.691,Z 759.497,A -85,B 0,C 180,E1 13439.855,E2 13439.855} C_VEL
LIN {X 0,Y 272.563,Z 768.875,A -85,B 0,C 180,E1 13435.883,E2 13435.883} C_VEL
LIN {X 0,Y 269.267,Z 776.816,A -85,B 0,C 180,E1 13431.569,E2 13431.569} C_VEL
LIN {X 0,Y 267.002,Z 782.843,A -85,B 0,C 180,E1 13427.208,E2 13427.208} C_VEL
LIN {X 0,Y 265.652,Z 787.091,A -85,B 0,C 180,E1 13422.83,E2 13422.83} C_VEL
LIN {X 0,Y 264.971,Z 789.663,A -85,B 0,C 180,E1 13418.463,E2 13418.463} C_VEL
LIN {X 0,Y 264.729,Z 790.612,A -85,B 0,C 180,E1 13414.332,E2 13414.332} C_VEL
LIN {X 0,Y 264.745,Z 790.148,A -85,B 0,C 180,E1 13410.216,E2 13410.216} C_VEL
LIN {X 0,Y 265.042,Z 788.28,A -85,B 0,C 180,E1 13406.106,E2 13406.106} C_VEL
LIN {X 0,Y 265.772,Z 784.981,A -85,B 0,C 180,E1 13401.999,E2 13401.999} C_VEL
LIN {X 0,Y 267.203,Z 779.859,A -85,B 0,C 180,E1 13397.685,E2 13397.685} C_VEL
LIN {X 0,Y 269.524,Z 772.942,A -85,B 0,C 180,E1 13393.402,E2 13393.402} C_VEL
LIN {X 0,Y 272.643,Z 764.583,A -85,B 0,C 180,E1 13389.387,E2 13389.387} C_VEL
LIN {X 0,Y 276.729,Z 754.241,A -85,B 0,C 180,E1 13385.448,E2 13385.448} C_VEL
LIN {X 0,Y 281.514,Z 742.364,A -85,B 0,C 180,E1 13381.811,E2 13381.811} C_VEL
LIN {X 0,Y 286.515,Z 729.816,A -85,B 0,C 180,E1 13378.67,E2 13378.67} C_VEL
LIN {X 0,Y 288.738,Z 724.137,A -85,B 0,C 180,E1 13377.423,E2 13377.423} C_VEL
LIN {X 0,Y 289.869,Z 719.122,A -85,B 0,C 180,E1 13376.277,E2 13376.277} C_VEL
LIN {X 0,Y 290.068,Z 706.512,A -85,B 0,C 180,E1 13373.172,E2 13373.172} C_VEL
LIN {X 0,Y 291.328,Z 700.92,A -85,B 0,C 180,E1 13372.144,E2 13372.144} C_VEL
LIN {X 0,Y 296.852,Z 684.734,A -85,B 0,C 180,E1 13369.871,E2 13369.871} C_VEL
LIN {X 0,Y 302.081,Z 667.645,A -85,B 0,C 180,E1 13367.913,E2 13367.913} C_VEL
LIN {X 0,Y 307.044,Z 648.852,A -85,B 0,C 180,E1 13366.179,E2 13366.179} C_VEL
LIN {X 0,Y 311.4,Z 628.802,A -85,B 0,C 180,E1 13364.726,E2 13364.726} C_VEL
LIN {X 0,Y 314.749,Z 609.044,A -85,B 0,C 180,E1 13363.631,E2 13363.631} C_VEL
LIN {X 0,Y 320.392,Z 570.466,A -85,B 0,C 180,E1 13362.051,E2 13362.051} C_VEL
LIN {X 0,Y 327.714,Z 518.191,A -85,B 0,C 180,E1 13360.36,E2 13360.36} C_VEL
LIN {X 0,Y 333.465,Z 467.841,A -85,B 0,C 180,E1 13358.982,E2 13358.982} C_VEL
LIN {X 0,Y 337.672,Z 418.555,A -85,B 0,C 180,E1 13357.862,E2 13357.862} C_VEL
LIN {X 0,Y 337.952,Z 414.212,A -85,B 0,C 180,E1 13357.766,E2 13357.766} C_VEL
LIN {X 0,Y 328.236,Z 424.441,A -85,B 0,C 180,E1 13355.526,E2 13355.526} C_VEL
LIN {X 0,Y 326.27,Z 427.268,A -85,B 0,C 180,E1 13355.072,E2 13355.072} C_VEL
LIN {X 0,Y 320.455,Z 438.834,A -85,B 0,C 180,E1 13353.819,E2 13353.819} C_VEL
LIN {X 0,Y 315.521,Z 446.677,A -85,B 0,C 180,E1 13352.597,E2 13352.597} C_VEL
LIN {X 0,Y 314.081,Z 448.977,A -85,B 0,C 180,E1 13352.225,E2 13352.225} C_VEL
LIN {X 0,Y 308.253,Z 461.589,A -85,B 0,C 180,E1 13350.858,E2 13350.858} C_VEL
LIN {X 0,Y 303.762,Z 469.491,A -85,B 0,C 180,E1 13349.615,E2 13349.615} C_VEL
LIN {X 0,Y 301.946,Z 472.407,A -85,B 0,C 180,E1 13349.075,E2 13349.075} C_VEL
LIN {X 0,Y 298.128,Z 482.113,A -85,B 0,C 180,E1 13348.168,E2 13348.168} C_VEL
LIN {X 0,Y 294.061,Z 495.213,A -85,B 0,C 180,E1 13347.435,E2 13347.435} C_VEL
LIN {X 0,Y 291.112,Z 502.439,A -85,B 0,C 180,E1 13346.706,E2 13346.706} C_VEL
LIN {X 0,Y 286.134,Z 520.385,A -85,B 0,C 180,E1 13346.082,E2 13346.082} C_VEL
LIN {X 0,Y 282.336,Z 531.558,A -85,B 0,C 180,E1 13345.388,E2 13345.388} C_VEL
LIN {X 0,Y 279.739,Z 537.535,A -85,B 0,C 180,E1 13344.693,E2 13344.693} C_VEL
LIN {X 0,Y 278.932,Z 539.233,A -85,B 0,C 180,E1 13344.459,E2 13344.459} C_VEL
LIN {X 0,Y 274.455,Z 553.642,A -85,B 0,C 180,E1 13343.893,E2 13343.893} C_VEL
LIN {X 0,Y 271.107,Z 562.639,A -85,B 0,C 180,E1 13343.215,E2 13343.215} C_VEL
LIN {X 0,Y 269.32,Z 566.243,A -85,B 0,C 180,E1 13342.656,E2 13342.656} C_VEL
LIN {X 0,Y 268.581,Z 567.118,A -85,B 0,C 180,E1 13342.274,E2 13342.274} C_VEL
LIN {X 0,Y 266.828,Z 620.12,A -85,B 0,C 180,E1 13340.21,E2 13340.21} C_VEL
LIN {X 0,Y 266.171,Z 638.477,A -85,B 0,C 180,E1 13339.169,E2 13339.169} C_VEL
LIN {X 0,Y 265.243,Z 655.752,A -85,B 0,C 180,E1 13337.779,E2 13337.779} C_VEL
LIN {X 0,Y 264.202,Z 671.229,A -85,B 0,C 180,E1 13336.151,E2 13336.151} C_VEL
LIN {X 0,Y 263,Z 686.736,A -85,B 0,C 180,E1 13334.083,E2 13334.083} C_VEL
LIN {X 0,Y 261.751,Z 701.609,A -85,B 0,C 180,E1 13331.57,E2 13331.57} C_VEL
LIN {X 0,Y 260.7,Z 714.492,A -85,B 0,C 180,E1 13328.825,E2 13328.825} C_VEL
LIN {X 0,Y 259.942,Z 725.259,A -85,B 0,C 180,E1 13325.962,E2 13325.962} C_VEL
LIN {X 0,Y 259.517,Z 733.96,A -85,B 0,C 180,E1 13323.093,E2 13323.093} C_VEL
LIN {X 0,Y 259.379,Z 741.718,A -85,B 0,C 180,E1 13319.78,E2 13319.78} C_VEL
LIN {X 0,Y 259.608,Z 747.052,A -85,B 0,C 180,E1 13316.689,E2 13316.689} C_VEL
LIN {X 0,Y 260.251,Z 750.98,A -85,B 0,C 180,E1 13313.382,E2 13313.382} C_VEL
LIN {X 0,Y 261.311,Z 753.02,A -85,B 0,C 180,E1 13310.086,E2 13310.086} C_VEL
LIN {X 0,Y 262.874,Z 753.285,A -85,B 0,C 180,E1 13306.809,E2 13306.809} C_VEL
LIN {X 0,Y 264.937,Z 751.656,A -85,B 0,C 180,E1 13303.559,E2 13303.559} C_VEL
LIN {X 0,Y 267.353,Z 748.448,A -85,B 0,C 180,E1 13300.559,E2 13300.559} C_VEL
LIN {X 0,Y 270.24,Z 743.385,A -85,B 0,C 180,E1 13297.6,E2 13297.6} C_VEL
LIN {X 0,Y 273.614,Z 736.355,A -85,B 0,C 180,E1 13294.689,E2 13294.689} C_VEL
LIN {X 0,Y 277.168,Z 727.754,A -85,B 0,C 180,E1 13292.034,E2 13292.034} C_VEL
LIN {X 0,Y 281.177,Z 716.49,A -85,B 0,C 180,E1 13289.379,E2 13289.379} C_VEL
LIN {X 0,Y 285.232,Z 703.235,A -85,B 0,C 180,E1 13286.97,E2 13286.97} C_VEL
LIN {X 0,Y 288.948,Z 688.943,A -85,B 0,C 180,E1 13284.942,E2 13284.942} C_VEL
LIN {X 0,Y 290.454,Z 682.62,A -85,B 0,C 180,E1 13284.183,E2 13284.183} C_VEL
LIN {X 0,Y 294.152,Z 680.667,A -85,B 0,C 180,E1 13283.668,E2 13283.668} C_VEL
LIN {X 0,Y 298.997,Z 676.487,A -85,B 0,C 180,E1 13283.232,E2 13283.232} C_VEL
LIN {X 0,Y 303.794,Z 672.977,A -85,B 0,C 180,E1 13282.73,E2 13282.73} C_VEL
LIN {X 0,Y 308.13,Z 668.748,A -85,B 0,C 180,E1 13282.408,E2 13282.408} C_VEL
LIN {X 0,Y 310.549,Z 666.896,A -85,B 0,C 180,E1 13282.178,E2 13282.178} C_VEL
LIN {X 0,Y 304.046,Z 692.298,A -85,B 0,C 180,E1 13280.163,E2 13280.163} C_VEL
LIN {X 0,Y 298.68,Z 711.572,A -85,B 0,C 180,E1 13278.29,E2 13278.29} C_VEL
LIN {X 0,Y 293.068,Z 729.08,A -85,B 0,C 180,E1 13276.167,E2 13276.167} C_VEL
LIN {X 0,Y 286.867,Z 746.651,A -85,B 0,C 180,E1 13273.534,E2 13273.534} C_VEL
LIN {X 0,Y 280.91,Z 762.3,A -85,B 0,C 180,E1 13270.645,E2 13270.645} C_VEL
LIN {X 0,Y 275.125,Z 776.781,A -85,B 0,C 180,E1 13267.367,E2 13267.367} C_VEL
LIN {X 0,Y 269.868,Z 789.816,A -85,B 0,C 180,E1 13263.763,E2 13263.763} C_VEL
LIN {X 0,Y 265.293,Z 801.356,A -85,B 0,C 180,E1 13259.834,E2 13259.834} C_VEL
LIN {X 0,Y 261.417,Z 811.936,A -85,B 0,C 180,E1 13255.365,E2 13255.365} C_VEL
LIN {X 0,Y 258.747,Z 820.431,A -85,B 0,C 180,E1 13250.825,E2 13250.825} C_VEL
LIN {X 0,Y 257.112,Z 827.354,A -85,B 0,C 180,E1 13246.028,E2 13246.028} C_VEL
LIN {X 0,Y 256.463,Z 832.234,A -85,B 0,C 180,E1 13241.469,E2 13241.469} C_VEL
LIN {X 0,Y 256.413,Z 835.456,A -85,B 0,C 180,E1 13236.943,E2 13236.943} C_VEL
LIN {X 0,Y 256.542,Z 837.102,A -85,B 0,C 180,E1 13232.681,E2 13232.681} C_VEL
LIN {X 0,Y 256.56,Z 837.404,A -85,B 0,C 180,E1 13228.66,E2 13228.66} C_VEL
LIN {X 0,Y 256.425,Z 836.404,A -85,B 0,C 180,E1 13224.406,E2 13224.406} C_VEL
LIN {X 0,Y 256.369,Z 833.892,A -85,B 0,C 180,E1 13219.892,E2 13219.892} C_VEL
LIN {X 0,Y 256.806,Z 829.847,A -85,B 0,C 180,E1 13215.34,E2 13215.34} C_VEL
LIN {X 0,Y 258.165,Z 823.829,A -85,B 0,C 180,E1 13210.544,E2 13210.544} C_VEL
LIN {X 0,Y 260.687,Z 815.964,A -85,B 0,C 180,E1 13205.77,E2 13205.77} C_VEL
LIN {X 0,Y 264.321,Z 806.478,A -85,B 0,C 180,E1 13201.288,E2 13201.288} C_VEL
LIN {X 0,Y 269.234,Z 794.873,A -85,B 0,C 180,E1 13196.912,E2 13196.912} C_VEL
LIN {X 0,Y 274.758,Z 782.23,A -85,B 0,C 180,E1 13193.098,E2 13193.098} C_VEL
LIN {X 0,Y 281.033,Z 767.877,A -85,B 0,C 180,E1 13189.584,E2 13189.584} C_VEL
LIN {X 0,Y 287.347,Z 752.848,A -85,B 0,C 180,E1 13186.589,E2 13186.589} C_VEL
LIN {X 0,Y 294.22,Z 735.309,A -85,B 0,C 180,E1 13183.767,E2 13183.767} C_VEL
LIN {X 0,Y 300.434,Z 717.905,A -85,B 0,C 180,E1 13181.512,E2 13181.512} C_VEL
LIN {X 0,Y 306.227,Z 699.495,A -85,B 0,C 180,E1 13179.595,E2 13179.595} C_VEL
LIN {X 0,Y 313.207,Z 674.146,A -85,B 0,C 180,E1 13177.505,E2 13177.505} C_VEL
LIN {X 0,Y 319.714,Z 648.477,A -85,B 0,C 180,E1 13175.821,E2 13175.821} C_VEL
LIN {X 0,Y 325.761,Z 622.213,A -85,B 0,C 180,E1 13174.474,E2 13174.474} C_VEL
LIN {X 0,Y 331.493,Z 592.897,A -85,B 0,C 180,E1 13173.314,E2 13173.314} C_VEL
LIN {X 0,Y 335.345,Z 569.457,A -85,B 0,C 180,E1 13172.616,E2 13172.616} C_VEL
LIN {X 0,Y 339.43,Z 545.603,A -85,B 0,C 180,E1 13172.302,E2 13172.302} C_VEL
LIN {X 0,Y 339.802,Z 542.846,A -85,B 0,C 180,E1 13172.259,E2 13172.259} C_VEL
LIN {X 0,Y 337.391,Z 536.152,A -85,B 0,C 180,E1 13171.338,E2 13171.338} C_VEL
LIN {X 0,Y 330.484,Z 549.48,A -85,B 0,C 180,E1 13170.172,E2 13170.172} C_VEL
LIN {X 0,Y 327.322,Z 555.953,A -85,B 0,C 180,E1 13169.691,E2 13169.691} C_VEL
LIN {X 0,Y 321.477,Z 572.813,A -85,B 0,C 180,E1 13169.216,E2 13169.216} C_VEL
LIN {X 0,Y 316.249,Z 584.341,A -85,B 0,C 180,E1 13168.644,E2 13168.644} C_VEL
LIN {X 0,Y 314.519,Z 587.928,A -85,B 0,C 180,E1 13168.447,E2 13168.447} C_VEL
LIN {X 0,Y 308.76,Z 601.391,A -85,B 0,C 180,E1 13168.021,E2 13168.021} C_VEL
LIN {X 0,Y 304.003,Z 609.897,A -85,B 0,C 180,E1 13167.469,E2 13167.469} C_VEL
LIN {X 0,Y 301.961,Z 614.193,A -85,B 0,C 180,E1 13167.319,E2 13167.319} C_VEL
LIN {X 0,Y 297.196,Z 623.489,A -85,B 0,C 180,E1 13166.931,E2 13166.931} C_VEL
LIN {X 0,Y 292.714,Z 630.405,A -85,B 0,C 180,E1 13166.362,E2 13166.362} C_VEL
LIN {X 0,Y 288.823,Z 637.792,A -85,B 0,C 180,E1 13166.081,E2 13166.081} C_VEL
LIN {X 0,Y 285.408,Z 642.746,A -85,B 0,C 180,E1 13165.635,E2 13165.635} C_VEL
LIN {X 0,Y 284.019,Z 644.568,A -85,B 0,C 180,E1 13165.358,E2 13165.358} C_VEL
LIN {X 0,Y 282.508,Z 667.605,A -85,B 0,C 180,E1 13164.066,E2 13164.066} C_VEL
LIN {X 0,Y 281.101,Z 681.79,A -85,B 0,C 180,E1 13162.922,E2 13162.922} C_VEL
LIN {X 0,Y 279.15,Z 695.617,A -85,B 0,C 180,E1 13161.428,E2 13161.428} C_VEL
LIN {X 0,Y 276.961,Z 707.748,A -85,B 0,C 180,E1 13159.727,E2 13159.727} C_VEL
LIN {X 0,Y 274.557,Z 718.41,A -85,B 0,C 180,E1 13157.812,E2 13157.812} C_VEL
LIN {X 0,Y 271.956,Z 728.2,A -85,B 0,C 180,E1 13155.568,E2 13155.568} C_VEL
LIN {X 0,Y 269.338,Z 736.388,A -85,B 0,C 180,E1 13153.087,E2 13153.087} C_VEL
LIN {X 0,Y 266.826,Z 743.021,A -85,B 0,C 180,E1 13150.361,E2 13150.361} C_VEL
LIN {X 0,Y 264.664,Z 747.619,A -85,B 0,C 180,E1 13147.597,E2 13147.597} C_VEL
LIN {X 0,Y 262.869,Z 750.54,A -85,B 0,C 180,E1 13144.75,E2 13144.75} C_VEL
LIN {X 0,Y 261.409,Z 751.736,A -85,B 0,C 180,E1 13141.753,E2 13141.753} C_VEL
LIN {X 0,Y 260.346,Z 751.096,A -85,B 0,C 180,E1 13138.679,E2 13138.679} C_VEL
LIN {X 0,Y 259.696,Z 748.739,A -85,B 0,C 180,E1 13135.702,E2 13135.702} C_VEL
LIN {X 0,Y 259.398,Z 744.593,A -85,B 0,C 180,E1 13132.691,E2 13132.691} C_VEL
LIN {X 0,Y 259.443,Z 738.216,A -85,B 0,C 180,E1 13129.563,E2 13129.563} C_VEL
LIN {X 0,Y 259.813,Z 730.103,A -85,B 0,C 180,E1 13126.649,E2 13126.649} C_VEL
LIN {X 0,Y 260.462,Z 720.35,A -85,B 0,C 180,E1 13123.954,E2 13123.954} C_VEL
LIN {X 0,Y 261.349,Z 708.358,A -85,B 0,C 180,E1 13121.369,E2 13121.369} C_VEL
LIN {X 0,Y 262.327,Z 694.92,A -85,B 0,C 180,E1 13119.121,E2 13119.121} C_VEL
LIN {X 0,Y 263.21,Z 681.125,A -85,B 0,C 180,E1 13117.332,E2 13117.332} C_VEL
LIN {X 0,Y 263.982,Z 666.074,A -85,B 0,C 180,E1 13115.853,E2 13115.853} C_VEL
LIN {X 0,Y 264.296,Z 659.194,A -85,B 0,C 180,E1 13115.289,E2 13115.289} C_VEL
LIN {X 0,Y 265.343,Z 659.248,A -85,B 0,C 180,E1 13114.739,E2 13114.739} C_VEL
LIN {X 0,Y 267.676,Z 657.282,A -85,B 0,C 180,E1 13114.084,E2 13114.084} C_VEL
LIN {X 0,Y 270.736,Z 653.353,A -85,B 0,C 180,E1 13113.574,E2 13113.574} C_VEL
LIN {X 0,Y 272.275,Z 651.122,A -85,B 0,C 180,E1 13113.383,E2 13113.383} C_VEL
LIN {X 0,Y 274.774,Z 649.008,A -85,B 0,C 180,E1 13112.709,E2 13112.709} C_VEL
LIN {X 0,Y 277.972,Z 645.098,A -85,B 0,C 180,E1 13112.12,E2 13112.12} C_VEL
LIN {X 0,Y 281.918,Z 638.681,A -85,B 0,C 180,E1 13111.686,E2 13111.686} C_VEL
LIN {X 0,Y 282.688,Z 637.397,A -85,B 0,C 180,E1 13111.593,E2 13111.593} C_VEL
LIN {X 0,Y 286.446,Z 632.832,A -85,B 0,C 180,E1 13110.86,E2 13110.86} C_VEL
LIN {X 0,Y 290.668,Z 625.853,A -85,B 0,C 180,E1 13110.307,E2 13110.307} C_VEL
LIN {X 0,Y 294.057,Z 618.99,A -85,B 0,C 180,E1 13109.982,E2 13109.982} C_VEL
LIN {X 0,Y 298.366,Z 612.617,A -85,B 0,C 180,E1 13109.238,E2 13109.238} C_VEL
LIN {X 0,Y 302.876,Z 603.829,A -85,B 0,C 180,E1 13108.692,E2 13108.692} C_VEL
LIN {X 0,Y 306.023,Z 596.81,A -85,B 0,C 180,E1 13108.399,E2 13108.399} C_VEL
LIN {X 0,Y 310.739,Z 589.003,A -85,B 0,C 180,E1 13107.673,E2 13107.673} C_VEL
LIN {X 0,Y 315.638,Z 578.593,A -85,B 0,C 180,E1 13107.147,E2 13107.147} C_VEL
LIN {X 0,Y 318.417,Z 571.939,A -85,B 0,C 180,E1 13106.907,E2 13106.907} C_VEL
LIN {X 0,Y 323.447,Z 562.937,A -85,B 0,C 180,E1 13106.203,E2 13106.203} C_VEL
LIN {X 0,Y 328.645,Z 550.917,A -85,B 0,C 180,E1 13105.681,E2 13105.681} C_VEL
LIN {X 0,Y 330.349,Z 546.791,A -85,B 0,C 180,E1 13105.528,E2 13105.528} C_VEL
LIN {X 0,Y 322.696,Z 596.492,A -85,B 0,C 180,E1 13103.739,E2 13103.739} C_VEL
LIN {X 0,Y 318.766,Z 620.866,A -85,B 0,C 180,E1 13102.595,E2 13102.595} C_VEL
LIN {X 0,Y 314.507,Z 641.214,A -85,B 0,C 180,E1 13101.305,E2 13101.305} C_VEL
LIN {X 0,Y 309.394,Z 660.817,A -85,B 0,C 180,E1 13099.701,E2 13099.701} C_VEL
LIN {X 0,Y 303.702,Z 679.244,A -85,B 0,C 180,E1 13097.796,E2 13097.796} C_VEL
LIN {X 0,Y 297.56,Z 696.606,A -85,B 0,C 180,E1 13095.565,E2 13095.565} C_VEL
LIN {X 0,Y 291.16,Z 712.794,A -85,B 0,C 180,E1 13092.99,E2 13092.99} C_VEL
LIN {X 0,Y 284.7,Z 727.825,A -85,B 0,C 180,E1 13090.037,E2 13090.037} C_VEL
LIN {X 0,Y 278.638,Z 741.127,A -85,B 0,C 180,E1 13086.817,E2 13086.817} C_VEL
LIN {X 0,Y 273.099,Z 752.876,A -85,B 0,C 180,E1 13083.311,E2 13083.311} C_VEL
LIN {X 0,Y 268.187,Z 763.228,A -85,B 0,C 180,E1 13079.481,E2 13079.481} C_VEL
LIN {X 0,Y 264.065,Z 772.112,A -85,B 0,C 180,E1 13075.332,E2 13075.332} C_VEL
LIN {X 0,Y 260.863,Z 779.457,A -85,B 0,C 180,E1 13070.883,E2 13070.883} C_VEL
LIN {X 0,Y 258.641,Z 785.173,A -85,B 0,C 180,E1 13066.161,E2 13066.161} C_VEL
LIN {X 0,Y 257.453,Z 788.839,A -85,B 0,C 180,E1 13061.651,E2 13061.651} C_VEL
LIN {X 0,Y 256.898,Z 790.868,A -85,B 0,C 180,E1 13057.155,E2 13057.155} C_VEL
LIN {X 0,Y 256.739,Z 791.334,A -85,B 0,C 180,E1 13052.902,E2 13052.902} C_VEL
LIN {X 0,Y 256.861,Z 790.395,A -85,B 0,C 180,E1 13048.662,E2 13048.662} C_VEL
LIN {X 0,Y 257.356,Z 787.863,A -85,B 0,C 180,E1 13044.203,E2 13044.203} C_VEL
LIN {X 0,Y 258.456,Z 783.697,A -85,B 0,C 180,E1 13039.749,E2 13039.749} C_VEL
LIN {X 0,Y 260.391,Z 777.814,A -85,B 0,C 180,E1 13035.319,E2 13035.319} C_VEL
LIN {X 0,Y 263.312,Z 770.087,A -85,B 0,C 180,E1 13030.94,E2 13030.94} C_VEL
LIN {X 0,Y 267.091,Z 760.858,A -85,B 0,C 180,E1 13026.854,E2 13026.854} C_VEL
LIN {X 0,Y 271.606,Z 750.199,A -85,B 0,C 180,E1 13023.077,E2 13023.077} C_VEL
LIN {X 0,Y 276.718,Z 738.15,A -85,B 0,C 180,E1 13019.611,E2 13019.611} C_VEL
LIN {X 0,Y 282.256,Z 724.699,A -85,B 0,C 180,E1 13016.453,E2 13016.453} C_VEL
LIN {X 0,Y 288.073,Z 709.791,A -85,B 0,C 180,E1 13013.593,E2 13013.593} C_VEL
LIN {X 0,Y 291.328,Z 700.92,A -85,B 0,C 180,E1 13012.144,E2 13012.144} C_VEL
LIN {X 0,Y 292.624,Z 695.274,A -85,B 0,C 180,E1 13011.147,E2 13011.147} C_VEL
LIN {X 0,Y 293.242,Z 680.961,A -85,B 0,C 180,E1 13008.381,E2 13008.381} C_VEL
LIN {X 0,Y 294.529,Z 674.694,A -85,B 0,C 180,E1 13007.512,E2 13007.512} C_VEL
LIN {X 0,Y 299.54,Z 657.433,A -85,B 0,C 180,E1 13005.762,E2 13005.762} C_VEL
LIN {X 0,Y 303.938,Z 639.696,A -85,B 0,C 180,E1 13004.315,E2 13004.315} C_VEL
LIN {X 0,Y 307.744,Z 620.823,A -85,B 0,C 180,E1 13003.096,E2 13003.096} C_VEL
LIN {X 0,Y 311.621,Z 596.274,A -85,B 0,C 180,E1 13001.91,E2 13001.91} C_VEL
LIN {X 0,Y 318.317,Z 552.536,A -85,B 0,C 180,E1 13000.28,E2 13000.28} C_VEL
LIN {X 0,Y 325.236,Z 501.769,A -85,B 0,C 180,E1 12998.722,E2 12998.722} C_VEL
LIN {X 0,Y 330.593,Z 451.994,A -85,B 0,C 180,E1 12997.445,E2 12997.445} C_VEL
LIN {X 0,Y 332.595,Z 428.148,A -85,B 0,C 180,E1 12996.906,E2 12996.906} C_VEL
LIN {X 0,Y 329.448,Z 431.558,A -85,B 0,C 180,E1 12996.179,E2 12996.179} C_VEL
LIN {X 0,Y 321.902,Z 445.6,A -85,B 0,C 180,E1 12994.614,E2 12994.614} C_VEL
LIN {X 0,Y 316.731,Z 453.366,A -85,B 0,C 180,E1 12993.373,E2 12993.373} C_VEL
LIN {X 0,Y 309.814,Z 467.577,A -85,B 0,C 180,E1 12991.821,E2 12991.821} C_VEL
LIN {X 0,Y 304.967,Z 475.674,A -85,B 0,C 180,E1 12990.544,E2 12990.544} C_VEL
LIN {X 0,Y 303.631,Z 477.885,A -85,B 0,C 180,E1 12990.173,E2 12990.173} C_VEL
LIN {X 0,Y 300.565,Z 485.417,A -85,B 0,C 180,E1 12989.495,E2 12989.495} C_VEL
LIN {X 0,Y 296.21,Z 498.872,A -85,B 0,C 180,E1 12988.752,E2 12988.752} C_VEL
LIN {X 0,Y 293.149,Z 506.6,A -85,B 0,C 180,E1 12988.08,E2 12988.08} C_VEL
LIN {X 0,Y 288.154,Z 523.789,A -85,B 0,C 180,E1 12987.484,E2 12987.484} C_VEL
LIN {X 0,Y 284.14,Z 535.164,A -85,B 0,C 180,E1 12986.785,E2 12986.785} C_VEL
LIN {X 0,Y 280.98,Z 542.142,A -85,B 0,C 180,E1 12986.014,E2 12986.014} C_VEL
LIN {X 0,Y 279.667,Z 546.215,A -85,B 0,C 180,E1 12985.832,E2 12985.832} C_VEL
LIN {X 0,Y 275.274,Z 559.347,A -85,B 0,C 180,E1 12985.235,E2 12985.235} C_VEL
LIN {X 0,Y 271.849,Z 567.727,A -85,B 0,C 180,E1 12984.53,E2 12984.53} C_VEL
LIN {X 0,Y 269.3,Z 572.684,A -85,B 0,C 180,E1 12983.786,E2 12983.786} C_VEL
LIN {X 0,Y 264.936,Z 585.185,A -85,B 0,C 180,E1 12983.228,E2 12983.228} C_VEL
LIN {X 0,Y 261.849,Z 592.187,A -85,B 0,C 180,E1 12982.567,E2 12982.567} C_VEL
LIN {X 0,Y 260.245,Z 594.942,A -85,B 0,C 180,E1 12982,E2 12982} C_VEL
LIN {X 0,Y 259.656,Z 595.451,A -85,B 0,C 180,E1 12981.644,E2 12981.644} C_VEL
LIN {X 0,Y 258.791,Z 628.719,A -85,B 0,C 180,E1 12980.187,E2 12980.187} C_VEL
LIN {X 0,Y 257.939,Z 647.532,A -85,B 0,C 180,E1 12978.898,E2 12978.898} C_VEL
LIN {X 0,Y 256.809,Z 665.225,A -85,B 0,C 180,E1 12977.212,E2 12977.212} C_VEL
LIN {X 0,Y 255.511,Z 682.239,A -85,B 0,C 180,E1 12975.084,E2 12975.084} C_VEL
LIN {X 0,Y 254.208,Z 697.72,A -85,B 0,C 180,E1 12972.61,E2 12972.61} C_VEL
LIN {X 0,Y 253.023,Z 711.735,A -85,B 0,C 180,E1 12969.784,E2 12969.784} C_VEL
LIN {X 0,Y 252.155,Z 723.397,A -85,B 0,C 180,E1 12966.833,E2 12966.833} C_VEL
LIN {X 0,Y 251.628,Z 732.741,A -85,B 0,C 180,E1 12963.874,E2 12963.874} C_VEL
LIN {X 0,Y 251.418,Z 740.722,A -85,B 0,C 180,E1 12960.684,E2 12960.684} C_VEL
LIN {X 0,Y 251.599,Z 747.144,A -85,B 0,C 180,E1 12957.267,E2 12957.267} C_VEL
LIN {X 0,Y 252.15,Z 751.408,A -85,B 0,C 180,E1 12954.083,E2 12954.083} C_VEL
LIN {X 0,Y 253.191,Z 754.144,A -85,B 0,C 180,E1 12950.683,E2 12950.683} C_VEL
LIN {X 0,Y 254.739,Z 755.111,A -85,B 0,C 180,E1 12947.303,E2 12947.303} C_VEL
LIN {X 0,Y 256.834,Z 754.199,A -85,B 0,C 180,E1 12943.955,E2 12943.955} C_VEL
LIN {X 0,Y 259.339,Z 751.674,A -85,B 0,C 180,E1 12940.836,E2 12940.836} C_VEL
LIN {X 0,Y 262.524,Z 747.088,A -85,B 0,C 180,E1 12937.614,E2 12937.614} C_VEL
LIN {X 0,Y 265.792,Z 741.353,A -85,B 0,C 180,E1 12934.845,E2 12934.845} C_VEL
LIN {X 0,Y 269.94,Z 732.827,A -85,B 0,C 180,E1 12931.831,E2 12931.831} C_VEL
LIN {X 0,Y 274.284,Z 722.371,A -85,B 0,C 180,E1 12929.071,E2 12929.071} C_VEL
LIN {X 0,Y 278.703,Z 710.174,A -85,B 0,C 180,E1 12926.587,E2 12926.587} C_VEL
LIN {X 0,Y 282.882,Z 696.767,A -85,B 0,C 180,E1 12924.449,E2 12924.449} C_VEL
LIN {X 0,Y 283.928,Z 693.472,A -85,B 0,C 180,E1 12923.979,E2 12923.979} C_VEL
LIN {X 0,Y 287.391,Z 691.894,A -85,B 0,C 180,E1 12923.482,E2 12923.482} C_VEL
LIN {X 0,Y 291.384,Z 688.749,A -85,B 0,C 180,E1 12923.095,E2 12923.095} C_VEL
LIN {X 0,Y 296.007,Z 685.971,A -85,B 0,C 180,E1 12922.555,E2 12922.555} C_VEL
LIN {X 0,Y 301.111,Z 681.826,A -85,B 0,C 180,E1 12922.114,E2 12922.114} C_VEL
LIN {X 0,Y 295.13,Z 703.459,A -85,B 0,C 180,E1 12920.186,E2 12920.186} C_VEL
LIN {X 0,Y 289.348,Z 721.597,A -85,B 0,C 180,E1 12918.146,E2 12918.146} C_VEL
LIN {X 0,Y 283.302,Z 738.768,A -85,B 0,C 180,E1 12915.762,E2 12915.762} C_VEL
LIN {X 0,Y 277.075,Z 754.897,A -85,B 0,C 180,E1 12913.003,E2 12913.003} C_VEL
LIN {X 0,Y 270.679,Z 770.457,A -85,B 0,C 180,E1 12909.721,E2 12909.721} C_VEL
LIN {X 0,Y 264.785,Z 784.382,A -85,B 0,C 180,E1 12906.092,E2 12906.092} C_VEL
LIN {X 0,Y 259.466,Z 796.941,A -85,B 0,C 180,E1 12902.031,E2 12902.031} C_VEL
LIN {X 0,Y 255.092,Z 807.868,A -85,B 0,C 180,E1 12897.648,E2 12897.648} C_VEL
LIN {X 0,Y 251.745,Z 817.259,A -85,B 0,C 180,E1 12892.865,E2 12892.865} C_VEL
LIN {X 0,Y 249.625,Z 824.764,A -85,B 0,C 180,E1 12887.964,E2 12887.964} C_VEL
LIN {X 0,Y 248.609,Z 830.35,A -85,B 0,C 180,E1 12883.016,E2 12883.016} C_VEL
LIN {X 0,Y 248.403,Z 834.034,A -85,B 0,C 180,E1 12878.332,E2 12878.332} C_VEL
LIN {X 0,Y 248.529,Z 836.086,A -85,B 0,C 180,E1 12873.922,E2 12873.922} C_VEL
LIN {X 0,Y 248.609,Z 836.743,A -85,B 0,C 180,E1 12869.769,E2 12869.769} C_VEL
LIN {X 0,Y 248.496,Z 836.172,A -85,B 0,C 180,E1 12865.615,E2 12865.615} C_VEL
LIN {X 0,Y 248.363,Z 834.253,A -85,B 0,C 180,E1 12861.2,E2 12861.2} C_VEL
LIN {X 0,Y 248.632,Z 830.709,A -85,B 0,C 180,E1 12856.512,E2 12856.512} C_VEL
LIN {X 0,Y 249.768,Z 825.296,A -85,B 0,C 180,E1 12851.564,E2 12851.564} C_VEL
LIN {X 0,Y 252.068,Z 818.072,A -85,B 0,C 180,E1 12846.63,E2 12846.63} C_VEL
LIN {X 0,Y 255.711,Z 808.748,A -85,B 0,C 180,E1 12841.762,E2 12841.762} C_VEL
LIN {X 0,Y 260.273,Z 798.419,A -85,B 0,C 180,E1 12837.464,E2 12837.464} C_VEL
LIN {X 0,Y 265.712,Z 786.597,A -85,B 0,C 180,E1 12833.519,E2 12833.519} C_VEL
LIN {X 0,Y 272.218,Z 772.538,A -85,B 0,C 180,E1 12829.725,E2 12829.725} C_VEL
LIN {X 0,Y 278.879,Z 757.678,A -85,B 0,C 180,E1 12826.498,E2 12826.498} C_VEL
LIN {X 0,Y 285.822,Z 741.171,A -85,B 0,C 180,E1 12823.603,E2 12823.603} C_VEL
LIN {X 0,Y 292.585,Z 723.646,A -85,B 0,C 180,E1 12821.121,E2 12821.121} C_VEL
LIN {X 0,Y 299.078,Z 704.694,A -85,B 0,C 180,E1 12818.987,E2 12818.987} C_VEL
LIN {X 0,Y 305.028,Z 684.711,A -85,B 0,C 180,E1 12817.199,E2 12817.199} C_VEL
LIN {X 0,Y 311.937,Z 659.088,A -85,B 0,C 180,E1 12815.343,E2 12815.343} C_VEL
LIN {X 0,Y 318.774,Z 631.357,A -85,B 0,C 180,E1 12813.778,E2 12813.778} C_VEL
LIN {X 0,Y 324.888,Z 603.059,A -85,B 0,C 180,E1 12812.561,E2 12812.561} C_VEL
LIN {X 0,Y 329.991,Z 574.148,A -85,B 0,C 180,E1 12811.591,E2 12811.591} C_VEL
LIN {X 0,Y 333.51,Z 553.724,A -85,B 0,C 180,E1 12811.219,E2 12811.219} C_VEL
LIN {X 0,Y 330.795,Z 559.205,A -85,B 0,C 180,E1 12810.835,E2 12810.835} C_VEL
LIN {X 0,Y 324.781,Z 576.075,A -85,B 0,C 180,E1 12810.374,E2 12810.374} C_VEL
LIN {X 0,Y 319.229,Z 588.018,A -85,B 0,C 180,E1 12809.808,E2 12809.808} C_VEL
LIN {X 0,Y 317.62,Z 591.444,A -85,B 0,C 180,E1 12809.652,E2 12809.652} C_VEL
LIN {X 0,Y 311.625,Z 604.956,A -85,B 0,C 180,E1 12809.236,E2 12809.236} C_VEL
LIN {X 0,Y 305.984,Z 615.008,A -85,B 0,C 180,E1 12808.652,E2 12808.652} C_VEL
LIN {X 0,Y 300.696,Z 625.537,A -85,B 0,C 180,E1 12808.293,E2 12808.293} C_VEL
LIN {X 0,Y 296.054,Z 632.702,A -85,B 0,C 180,E1 12807.778,E2 12807.778} C_VEL
LIN {X 0,Y 289.982,Z 643.281,A -85,B 0,C 180,E1 12807.295,E2 12807.295} C_VEL
LIN {X 0,Y 285.901,Z 648.703,A -85,B 0,C 180,E1 12806.752,E2 12806.752} C_VEL
LIN {X 0,Y 281.846,Z 655.476,A -85,B 0,C 180,E1 12806.436,E2 12806.436} C_VEL
LIN {X 0,Y 278.595,Z 659.529,A -85,B 0,C 180,E1 12805.966,E2 12805.966} C_VEL
LIN {X 0,Y 277.751,Z 660.651,A -85,B 0,C 180,E1 12805.778,E2 12805.778} C_VEL
LIN {X 0,Y 276.397,Z 676.133,A -85,B 0,C 180,E1 12804.696,E2 12804.696} C_VEL
LIN {X 0,Y 274.279,Z 691.722,A -85,B 0,C 180,E1 12803.184,E2 12803.184} C_VEL
LIN {X 0,Y 271.872,Z 704.887,A -85,B 0,C 180,E1 12801.475,E2 12801.475} C_VEL
LIN {X 0,Y 269.068,Z 717.023,A -85,B 0,C 180,E1 12799.425,E2 12799.425} C_VEL
LIN {X 0,Y 266.296,Z 726.97,A -85,B 0,C 180,E1 12797.254,E2 12797.254} C_VEL
LIN {X 0,Y 263.359,Z 735.819,A -85,B 0,C 180,E1 12794.735,E2 12794.735} C_VEL
LIN {X 0,Y 260.509,Z 743.006,A -85,B 0,C 180,E1 12791.961,E2 12791.961} C_VEL
LIN {X 0,Y 257.857,Z 748.454,A -85,B 0,C 180,E1 12788.922,E2 12788.922} C_VEL
LIN {X 0,Y 255.668,Z 751.793,A -85,B 0,C 180,E1 12785.835,E2 12785.835} C_VEL
LIN {X 0,Y 253.953,Z 753.222,A -85,B 0,C 180,E1 12782.707,E2 12782.707} C_VEL
LIN {X 0,Y 252.705,Z 752.81,A -85,B 0,C 180,E1 12779.546,E2 12779.546} C_VEL
LIN {X 0,Y 251.889,Z 750.54,A -85,B 0,C 180,E1 12776.358,E2 12776.358} C_VEL
LIN {X 0,Y 251.48,Z 746.331,A -85,B 0,C 180,E1 12773.149,E2 12773.149} C_VEL
LIN {X 0,Y 251.449,Z 740.567,A -85,B 0,C 180,E1 12770.154,E2 12770.154} C_VEL
LIN {X 0,Y 251.76,Z 732.756,A -85,B 0,C 180,E1 12767.149,E2 12767.149} C_VEL
LIN {X 0,Y 252.296,Z 724.244,A -85,B 0,C 180,E1 12764.601,E2 12764.601} C_VEL
LIN {X 0,Y 253.135,Z 712.897,A -85,B 0,C 180,E1 12761.936,E2 12761.936} C_VEL
LIN {X 0,Y 254.075,Z 700.319,A -85,B 0,C 180,E1 12759.617,E2 12759.617} C_VEL
LIN {X 0,Y 255.025,Z 686.66,A -85,B 0,C 180,E1 12757.647,E2 12757.647} C_VEL
LIN {X 0,Y 255.869,Z 672.094,A -85,B 0,C 180,E1 12756.02,E2 12756.02} C_VEL
LIN {X 0,Y 256.956,Z 672.161,A -85,B 0,C 180,E1 12755.394,E2 12755.394} C_VEL
LIN {X 0,Y 259.379,Z 670.319,A -85,B 0,C 180,E1 12754.666,E2 12754.666} C_VEL
LIN {X 0,Y 262.795,Z 666.443,A -85,B 0,C 180,E1 12754.052,E2 12754.052} C_VEL
LIN {X 0,Y 266.575,Z 663.533,A -85,B 0,C 180,E1 12753.009,E2 12753.009} C_VEL
LIN {X 0,Y 270.323,Z 659.445,A -85,B 0,C 180,E1 12752.341,E2 12752.341} C_VEL
LIN {X 0,Y 272.628,Z 656.501,A -85,B 0,C 180,E1 12752.001,E2 12752.001} C_VEL
LIN {X 0,Y 276.28,Z 653.022,A -85,B 0,C 180,E1 12751.227,E2 12751.227} C_VEL
LIN {X 0,Y 280.318,Z 647.979,A -85,B 0,C 180,E1 12750.629,E2 12750.629} C_VEL
LIN {X 0,Y 284.087,Z 642.023,A -85,B 0,C 180,E1 12750.246,E2 12750.246} C_VEL
LIN {X 0,Y 288.611,Z 636.546,A -85,B 0,C 180,E1 12749.5,E2 12749.5} C_VEL
LIN {X 0,Y 293.015,Z 629.495,A -85,B 0,C 180,E1 12748.984,E2 12748.984} C_VEL
LIN {X 0,Y 296.32,Z 623.197,A -85,B 0,C 180,E1 12748.691,E2 12748.691} C_VEL
LIN {X 0,Y 301.209,Z 615.968,A -85,B 0,C 180,E1 12747.946,E2 12747.946} C_VEL
LIN {X 0,Y 306.123,Z 606.409,A -85,B 0,C 180,E1 12747.403,E2 12747.403} C_VEL
LIN {X 0,Y 308.827,Z 600.626,A -85,B 0,C 180,E1 12747.159,E2 12747.159} C_VEL
LIN {X 0,Y 314.012,Z 591.986,A -85,B 0,C 180,E1 12746.437,E2 12746.437} C_VEL
LIN {X 0,Y 319.269,Z 580.787,A -85,B 0,C 180,E1 12745.918,E2 12745.918} C_VEL
LIN {X 0,Y 321.506,Z 575.663,A -85,B 0,C 180,E1 12745.725,E2 12745.725} C_VEL
LIN {X 0,Y 315.606,Z 611.895,A -85,B 0,C 180,E1 12744.236,E2 12744.236} C_VEL
LIN {X 0,Y 311.827,Z 631.795,A -85,B 0,C 180,E1 12743.132,E2 12743.132} C_VEL
LIN {X 0,Y 307.031,Z 651.532,A -85,B 0,C 180,E1 12741.705,E2 12741.705} C_VEL
LIN {X 0,Y 301.545,Z 670.173,A -85,B 0,C 180,E1 12739.992,E2 12739.992} C_VEL
LIN {X 0,Y 295.461,Z 687.9,A -85,B 0,C 180,E1 12737.957,E2 12737.957} C_VEL
LIN {X 0,Y 289.038,Z 704.508,A -85,B 0,C 180,E1 12735.59,E2 12735.59} C_VEL
LIN {X 0,Y 282.339,Z 720.156,A -85,B 0,C 180,E1 12732.839,E2 12732.839} C_VEL
LIN {X 0,Y 275.627,Z 734.661,A -85,B 0,C 180,E1 12729.677,E2 12729.677} C_VEL
LIN {X 0,Y 269.32,Z 747.574,A -85,B 0,C 180,E1 12726.178,E2 12726.178} C_VEL
LIN {X 0,Y 263.601,Z 758.957,A -85,B 0,C 180,E1 12722.332,E2 12722.332} C_VEL
LIN {X 0,Y 258.673,Z 768.799,A -85,B 0,C 180,E1 12718.137,E2 12718.137} C_VEL
LIN {X 0,Y 254.685,Z 777.054,A -85,B 0,C 180,E1 12713.606,E2 12713.606} C_VEL
LIN {X 0,Y 251.871,Z 783.374,A -85,B 0,C 180,E1 12708.997,E2 12708.997} C_VEL
LIN {X 0,Y 250.115,Z 787.906,A -85,B 0,C 180,E1 12704.351,E2 12704.351} C_VEL
LIN {X 0,Y 249.191,Z 790.753,A -85,B 0,C 180,E1 12699.702,E2 12699.702} C_VEL
LIN {X 0,Y 248.816,Z 791.999,A -85,B 0,C 180,E1 12695.072,E2 12695.072} C_VEL
LIN {X 0,Y 248.797,Z 791.739,A -85,B 0,C 180,E1 12690.691,E2 12690.691} C_VEL
LIN {X 0,Y 249.093,Z 790.082,A -85,B 0,C 180,E1 12686.318,E2 12686.318} C_VEL
LIN {X 0,Y 249.922,Z 786.766,A -85,B 0,C 180,E1 12681.719,E2 12681.719} C_VEL
LIN {X 0,Y 251.613,Z 781.482,A -85,B 0,C 180,E1 12676.908,E2 12676.908} C_VEL
LIN {X 0,Y 254.235,Z 774.632,A -85,B 0,C 180,E1 12672.373,E2 12672.373} C_VEL
LIN {X 0,Y 257.737,Z 766.344,A -85,B 0,C 180,E1 12668.135,E2 12668.135} C_VEL
LIN {X 0,Y 262.28,Z 756.088,A -85,B 0,C 180,E1 12663.998,E2 12663.998} C_VEL
LIN {X 0,Y 267.561,Z 744.304,A -85,B 0,C 180,E1 12660.197,E2 12660.197} C_VEL
LIN {X 0,Y 273.039,Z 731.854,A -85,B 0,C 180,E1 12656.932,E2 12656.932} C_VEL
LIN {X 0,Y 279.019,Z 717.608,A -85,B 0,C 180,E1 12653.88,E2 12653.88} C_VEL
LIN {X 0,Y 285.025,Z 702.327,A -85,B 0,C 180,E1 12651.205,E2 12651.205} C_VEL
LIN {X 0,Y 291.036,Z 685.43,A -85,B 0,C 180,E1 12648.798,E2 12648.798} C_VEL
LIN {X 0,Y 294.529,Z 674.694,A -85,B 0,C 180,E1 12647.512,E2 12647.512} C_VEL
LIN {X 0,Y 295.837,Z 668.378,A -85,B 0,C 180,E1 12646.669,E2 12646.669} C_VEL
LIN {X 0,Y 296.366,Z 653.496,A -85,B 0,C 180,E1 12644.383,E2 12644.383} C_VEL
LIN {X 0,Y 297.223,Z 646.785,A -85,B 0,C 180,E1 12643.655,E2 12643.655} C_VEL
LIN {X 0,Y 297.438,Z 645.78,A -85,B 0,C 180,E1 12643.575,E2 12643.575} C_VEL
LIN {X 0,Y 301.687,Z 626.597,A -85,B 0,C 180,E1 12642.242,E2 12642.242} C_VEL
LIN {X 0,Y 305.353,Z 605.233,A -85,B 0,C 180,E1 12641.12,E2 12641.12} C_VEL
LIN {X 0,Y 311.572,Z 566.209,A -85,B 0,C 180,E1 12639.558,E2 12639.558} C_VEL
LIN {X 0,Y 318.997,Z 516.166,A -85,B 0,C 180,E1 12637.946,E2 12637.946} C_VEL
LIN {X 0,Y 324.867,Z 466.825,A -85,B 0,C 180,E1 12636.613,E2 12636.613} C_VEL
LIN {X 0,Y 326.763,Z 446.601,A -85,B 0,C 180,E1 12636.113,E2 12636.113} C_VEL
LIN {X 0,Y 320.728,Z 456.301,A -85,B 0,C 180,E1 12634.813,E2 12634.813} C_VEL
LIN {X 0,Y 318.358,Z 459.857,A -85,B 0,C 180,E1 12634.262,E2 12634.262} C_VEL
LIN {X 0,Y 311.887,Z 472.695,A -85,B 0,C 180,E1 12632.888,E2 12632.888} C_VEL
LIN {X 0,Y 306.583,Z 481.339,A -85,B 0,C 180,E1 12631.564,E2 12631.564} C_VEL
LIN {X 0,Y 305.227,Z 483.705,A -85,B 0,C 180,E1 12631.225,E2 12631.225} C_VEL
LIN {X 0,Y 303.162,Z 488.71,A -85,B 0,C 180,E1 12630.8,E2 12630.8} C_VEL
LIN {X 0,Y 298.553,Z 502.404,A -85,B 0,C 180,E1 12630.06,E2 12630.06} C_VEL
LIN {X 0,Y 295.519,Z 509.967,A -85,B 0,C 180,E1 12629.457,E2 12629.457} C_VEL
LIN {X 0,Y 290.405,Z 526.995,A -85,B 0,C 180,E1 12628.874,E2 12628.874} C_VEL
LIN {X 0,Y 286.082,Z 538.757,A -85,B 0,C 180,E1 12628.168,E2 12628.168} C_VEL
LIN {X 0,Y 282.433,Z 546.964,A -85,B 0,C 180,E1 12627.374,E2 12627.374} C_VEL
LIN {X 0,Y 277.694,Z 560.988,A -85,B 0,C 180,E1 12626.801,E2 12626.801} C_VEL
LIN {X 0,Y 273.721,Z 570.712,A -85,B 0,C 180,E1 12626.068,E2 12626.068} C_VEL
LIN {X 0,Y 270.636,Z 576.87,A -85,B 0,C 180,E1 12625.304,E2 12625.304} C_VEL
LIN {X 0,Y 266.185,Z 588.963,A -85,B 0,C 180,E1 12624.74,E2 12624.74} C_VEL
LIN {X 0,Y 262.804,Z 596.515,A -85,B 0,C 180,E1 12624.023,E2 12624.023} C_VEL
LIN {X 0,Y 260.254,Z 600.746,A -85,B 0,C 180,E1 12623.239,E2 12623.239} C_VEL
LIN {X 0,Y 255.973,Z 611.628,A -85,B 0,C 180,E1 12622.629,E2 12622.629} C_VEL
LIN {X 0,Y 253.065,Z 617.488,A -85,B 0,C 180,E1 12621.925,E2 12621.925} C_VEL
LIN {X 0,Y 251.826,Z 619.287,A -85,B 0,C 180,E1 12621.426,E2 12621.426} C_VEL
LIN {X 0,Y 251.268,Z 619.67,A -85,B 0,C 180,E1 12621.048,E2 12621.048} C_VEL
LIN {X 0,Y 250.605,Z 637.923,A -85,B 0,C 180,E1 12620.007,E2 12620.007} C_VEL
LIN {X 0,Y 249.631,Z 655.577,A -85,B 0,C 180,E1 12618.569,E2 12618.569} C_VEL
LIN {X 0,Y 248.395,Z 673.073,A -85,B 0,C 180,E1 12616.66,E2 12616.66} C_VEL
LIN {X 0,Y 247.086,Z 689.06,A -85,B 0,C 180,E1 12614.411,E2 12614.411} C_VEL
LIN {X 0,Y 245.776,Z 704.088,A -85,B 0,C 180,E1 12611.737,E2 12611.737} C_VEL
LIN {X 0,Y 244.658,Z 717.561,A -85,B 0,C 180,E1 12608.698,E2 12608.698} C_VEL
LIN {X 0,Y 243.877,Z 729.108,A -85,B 0,C 180,E1 12605.412,E2 12605.412} C_VEL
LIN {X 0,Y 243.495,Z 738.229,A -85,B 0,C 180,E1 12602.119,E2 12602.119} C_VEL
LIN {X 0,Y 243.507,Z 745.34,A -85,B 0,C 180,E1 12598.824,E2 12598.824} C_VEL
LIN {X 0,Y 244.001,Z 751.253,A -85,B 0,C 180,E1 12595.064,E2 12595.064} C_VEL
LIN {X 0,Y 244.956,Z 754.821,A -85,B 0,C 180,E1 12591.551,E2 12591.551} C_VEL
LIN {X 0,Y 246.46,Z 756.633,A -85,B 0,C 180,E1 12588.06,E2 12588.06} C_VEL
LIN {X 0,Y 248.69,Z 756.505,A -85,B 0,C 180,E1 12584.374,E2 12584.374} C_VEL
LIN {X 0,Y 251.411,Z 754.521,A -85,B 0,C 180,E1 12580.968,E2 12580.968} C_VEL
LIN {X 0,Y 254.775,Z 750.648,A -85,B 0,C 180,E1 12577.625,E2 12577.625} C_VEL
LIN {X 0,Y 258.466,Z 745.122,A -85,B 0,C 180,E1 12574.572,E2 12574.572} C_VEL
LIN {X 0,Y 262.396,Z 738.281,A -85,B 0,C 180,E1 12571.804,E2 12571.804} C_VEL
LIN {X 0,Y 267.121,Z 728.68,A -85,B 0,C 180,E1 12568.9,E2 12568.9} C_VEL
LIN {X 0,Y 272.171,Z 716.859,A -85,B 0,C 180,E1 12566.183,E2 12566.183} C_VEL
LIN {X 0,Y 277.379,Z 703.391,A -85,B 0,C 180,E1 12563.761,E2 12563.761} C_VEL
LIN {X 0,Y 281.74,Z 701.43,A -85,B 0,C 180,E1 12563.148,E2 12563.148} C_VEL
LIN {X 0,Y 284.837,Z 699.495,A -85,B 0,C 180,E1 12562.829,E2 12562.829} C_VEL
LIN {X 0,Y 289.516,Z 696.866,A -85,B 0,C 180,E1 12562.267,E2 12562.267} C_VEL
LIN {X 0,Y 291.732,Z 695.243,A -85,B 0,C 180,E1 12562.076,E2 12562.076} C_VEL
LIN {X 0,Y 285.935,Z 713.971,A -85,B 0,C 180,E1 12560.135,E2 12560.135} C_VEL
LIN {X 0,Y 279.73,Z 731.557,A -85,B 0,C 180,E1 12557.875,E2 12557.875} C_VEL
LIN {X 0,Y 273.244,Z 748.078,A -85,B 0,C 180,E1 12555.226,E2 12555.226} C_VEL
LIN {X 0,Y 266.691,Z 763.708,A -85,B 0,C 180,E1 12552.152,E2 12552.152} C_VEL
LIN {X 0,Y 260.485,Z 777.809,A -85,B 0,C 180,E1 12548.732,E2 12548.732} C_VEL
LIN {X 0,Y 254.522,Z 791.131,A -85,B 0,C 180,E1 12544.724,E2 12544.724} C_VEL
LIN {X 0,Y 249.421,Z 802.832,A -85,B 0,C 180,E1 12540.338,E2 12540.338} C_VEL
LIN {X 0,Y 245.377,Z 812.859,A -85,B 0,C 180,E1 12535.59,E2 12535.59} C_VEL
LIN {X 0,Y 242.608,Z 821.017,A -85,B 0,C 180,E1 12530.688,E2 12530.688} C_VEL
LIN {X 0,Y 241.021,Z 827.358,A -85,B 0,C 180,E1 12525.643,E2 12525.643} C_VEL
LIN {X 0,Y 240.449,Z 831.99,A -85,B 0,C 180,E1 12520.543,E2 12520.543} C_VEL
LIN {X 0,Y 240.482,Z 834.665,A -85,B 0,C 180,E1 12515.966,E2 12515.966} C_VEL
LIN {X 0,Y 240.62,Z 835.892,A -85,B 0,C 180,E1 12511.667,E2 12511.667} C_VEL
LIN {X 0,Y 240.596,Z 835.895,A -85,B 0,C 180,E1 12507.618,E2 12507.618} C_VEL
LIN {X 0,Y 240.437,Z 834.714,A -85,B 0,C 180,E1 12503.313,E2 12503.313} C_VEL
LIN {X 0,Y 240.456,Z 831.965,A -85,B 0,C 180,E1 12498.487,E2 12498.487} C_VEL
LIN {X 0,Y 241.216,Z 827.367,A -85,B 0,C 180,E1 12493.381,E2 12493.381} C_VEL
LIN {X 0,Y 243.091,Z 821.008,A -85,B 0,C 180,E1 12488.273,E2 12488.273} C_VEL
LIN {X 0,Y 246.141,Z 813.139,A -85,B 0,C 180,E1 12483.459,E2 12483.459} C_VEL
LIN {X 0,Y 250.717,Z 802.932,A -85,B 0,C 180,E1 12478.586,E2 12478.586} C_VEL
LIN {X 0,Y 256.004,Z 791.99,A -85,B 0,C 180,E1 12474.412,E2 12474.412} C_VEL
LIN {X 0,Y 262.328,Z 779.055,A -85,B 0,C 180,E1 12470.467,E2 12470.467} C_VEL
LIN {X 0,Y 269.279,Z 764.556,A -85,B 0,C 180,E1 12466.904,E2 12466.904} C_VEL
LIN {X 0,Y 276.186,Z 749.434,A -85,B 0,C 180,E1 12463.91,E2 12463.91} C_VEL
LIN {X 0,Y 283.491,Z 732.147,A -85,B 0,C 180,E1 12461.148,E2 12461.148} C_VEL
LIN {X 0,Y 290.272,Z 714.384,A -85,B 0,C 180,E1 12458.879,E2 12458.879} C_VEL
LIN {X 0,Y 296.551,Z 695.517,A -85,B 0,C 180,E1 12456.957,E2 12456.957} C_VEL
LIN {X 0,Y 303.795,Z 670.513,A -85,B 0,C 180,E1 12454.963,E2 12454.963} C_VEL
LIN {X 0,Y 310.737,Z 644.342,A -85,B 0,C 180,E1 12453.3,E2 12453.3} C_VEL
LIN {X 0,Y 317.481,Z 616.161,A -85,B 0,C 180,E1 12451.923,E2 12451.923} C_VEL
LIN {X 0,Y 322.402,Z 591.556,A -85,B 0,C 180,E1 12450.958,E2 12450.958} C_VEL
LIN {X 0,Y 320.389,Z 596.02,A -85,B 0,C 180,E1 12450.81,E2 12450.81} C_VEL
LIN {X 0,Y 314.291,Z 609.171,A -85,B 0,C 180,E1 12450.399,E2 12450.399} C_VEL
LIN {X 0,Y 308.916,Z 618.559,A -85,B 0,C 180,E1 12449.897,E2 12449.897} C_VEL
LIN {X 0,Y 303.424,Z 629.138,A -85,B 0,C 180,E1 12449.546,E2 12449.546} C_VEL
LIN {X 0,Y 297.712,Z 637.985,A -85,B 0,C 180,E1 12448.988,E2 12448.988} C_VEL
LIN {X 0,Y 292.362,Z 647.02,A -85,B 0,C 180,E1 12448.606,E2 12448.606} C_VEL
LIN {X 0,Y 287.877,Z 653.128,A -85,B 0,C 180,E1 12448.09,E2 12448.09} C_VEL
LIN {X 0,Y 283.475,Z 659.937,A -85,B 0,C 180,E1 12447.747,E2 12447.747} C_VEL
LIN {X 0,Y 279.089,Z 665.413,A -85,B 0,C 180,E1 12447.179,E2 12447.179} C_VEL
LIN {X 0,Y 275.076,Z 671.082,A -85,B 0,C 180,E1 12446.789,E2 12446.789} C_VEL
LIN {X 0,Y 271.688,Z 674.492,A -85,B 0,C 180,E1 12446.206,E2 12446.206} C_VEL
LIN {X 0,Y 269.302,Z 690.555,A -85,B 0,C 180,E1 12444.688,E2 12444.688} C_VEL
LIN {X 0,Y 266.788,Z 703.546,A -85,B 0,C 180,E1 12443.056,E2 12443.056} C_VEL
LIN {X 0,Y 263.885,Z 715.676,A -85,B 0,C 180,E1 12441.097,E2 12441.097} C_VEL
LIN {X 0,Y 260.937,Z 725.706,A -85,B 0,C 180,E1 12439.007,E2 12439.007} C_VEL
LIN {X 0,Y 257.93,Z 734.52,A -85,B 0,C 180,E1 12436.669,E2 12436.669} C_VEL
LIN {X 0,Y 254.671,Z 742.41,A -85,B 0,C 180,E1 12433.856,E2 12433.856} C_VEL
LIN {X 0,Y 251.813,Z 748.186,A -85,B 0,C 180,E1 12430.986,E2 12430.986} C_VEL
LIN {X 0,Y 249.362,Z 752.053,A -85,B 0,C 180,E1 12428.067,E2 12428.067} C_VEL
LIN {X 0,Y 247.362,Z 754.281,A -85,B 0,C 180,E1 12425.101,E2 12425.101} C_VEL
LIN {X 0,Y 245.684,Z 754.817,A -85,B 0,C 180,E1 12421.865,E2 12421.865} C_VEL
LIN {X 0,Y 244.571,Z 753.684,A -85,B 0,C 180,E1 12418.828,E2 12418.828} C_VEL
LIN {X 0,Y 243.811,Z 750.666,A -85,B 0,C 180,E1 12415.53,E2 12415.53} C_VEL
LIN {X 0,Y 243.484,Z 745.688,A -85,B 0,C 180,E1 12412.211,E2 12412.211} C_VEL
LIN {X 0,Y 243.552,Z 739.08,A -85,B 0,C 180,E1 12409.114,E2 12409.114} C_VEL
LIN {X 0,Y 243.937,Z 731.047,A -85,B 0,C 180,E1 12406.246,E2 12406.246} C_VEL
LIN {X 0,Y 244.578,Z 721.694,A -85,B 0,C 180,E1 12403.615,E2 12403.615} C_VEL
LIN {X 0,Y 245.422,Z 710.691,A -85,B 0,C 180,E1 12401.143,E2 12401.143} C_VEL
LIN {X 0,Y 246.419,Z 697.627,A -85,B 0,C 180,E1 12398.83,E2 12398.83} C_VEL
LIN {X 0,Y 247.408,Z 683.519,A -85,B 0,C 180,E1 12396.856,E2 12396.856} C_VEL
LIN {X 0,Y 248.344,Z 683.549,A -85,B 0,C 180,E1 12396.258,E2 12396.258} C_VEL
LIN {X 0,Y 250.607,Z 682.112,A -85,B 0,C 180,E1 12395.484,E2 12395.484} C_VEL
LIN {X 0,Y 253.756,Z 679.05,A -85,B 0,C 180,E1 12394.814,E2 12394.814} C_VEL
LIN {X 0,Y 256.561,Z 677.425,A -85,B 0,C 180,E1 12393.871,E2 12393.871} C_VEL
LIN {X 0,Y 260.27,Z 674.128,A -85,B 0,C 180,E1 12393.043,E2 12393.043} C_VEL
LIN {X 0,Y 262.427,Z 671.891,A -85,B 0,C 180,E1 12392.669,E2 12392.669} C_VEL
LIN {X 0,Y 266.207,Z 668.994,A -85,B 0,C 180,E1 12391.754,E2 12391.754} C_VEL
LIN {X 0,Y 270.417,Z 664.642,A -85,B 0,C 180,E1 12391.028,E2 12391.028} C_VEL
LIN {X 0,Y 273.18,Z 661.5,A -85,B 0,C 180,E1 12390.629,E2 12390.629} C_VEL
LIN {X 0,Y 277.98,Z 656.835,A -85,B 0,C 180,E1 12389.763,E2 12389.763} C_VEL
LIN {X 0,Y 283.069,Z 650.299,A -85,B 0,C 180,E1 12389.13,E2 12389.13} C_VEL
LIN {X 0,Y 286.025,Z 646.101,A -85,B 0,C 180,E1 12388.844,E2 12388.844} C_VEL
LIN {X 0,Y 291.316,Z 639.525,A -85,B 0,C 180,E1 12388.091,E2 12388.091} C_VEL
LIN {X 0,Y 296.574,Z 631.127,A -85,B 0,C 180,E1 12387.584,E2 12387.584} C_VEL
LIN {X 0,Y 298.778,Z 627.156,A -85,B 0,C 180,E1 12387.398,E2 12387.398} C_VEL
LIN {X 0,Y 304.169,Z 619.27,A -85,B 0,C 180,E1 12386.675,E2 12386.675} C_VEL
LIN {X 0,Y 309.539,Z 609.067,A -85,B 0,C 180,E1 12386.149,E2 12386.149} C_VEL
LIN {X 0,Y 311.81,Z 604.382,A -85,B 0,C 180,E1 12385.946,E2 12385.946} C_VEL
LIN {X 0,Y 312.492,Z 603.485,A -85,B 0,C 180,E1 12385.838,E2 12385.838} C_VEL
LIN {X 0,Y 308.26,Z 626.852,A -85,B 0,C 180,E1 12384.663,E2 12384.663} C_VEL
LIN {X 0,Y 303.578,Z 646.769,A -85,B 0,C 180,E1 12383.321,E2 12383.321} C_VEL
LIN {X 0,Y 298.132,Z 665.585,A -85,B 0,C 180,E1 12381.701,E2 12381.701} C_VEL
LIN {X 0,Y 292.048,Z 683.421,A -85,B 0,C 180,E1 12379.771,E2 12379.771} C_VEL
LIN {X 0,Y 285.283,Z 700.734,A -85,B 0,C 180,E1 12377.434,E2 12377.434} C_VEL
LIN {X 0,Y 278.324,Z 716.693,A -85,B 0,C 180,E1 12374.759,E2 12374.759} C_VEL
LIN {X 0,Y 271.11,Z 731.859,A -85,B 0,C 180,E1 12371.594,E2 12371.594} C_VEL
LIN {X 0,Y 264.273,Z 745.353,A -85,B 0,C 180,E1 12368.076,E2 12368.076} C_VEL
LIN {X 0,Y 258.327,Z 756.648,A -85,B 0,C 180,E1 12364.409,E2 12364.409} C_VEL
LIN {X 0,Y 253.039,Z 766.578,A -85,B 0,C 180,E1 12360.383,E2 12360.383} C_VEL
LIN {X 0,Y 248.593,Z 775.076,A -85,B 0,C 180,E1 12356.003,E2 12356.003} C_VEL
LIN {X 0,Y 245.139,Z 782.064,A -85,B 0,C 180,E1 12351.285,E2 12351.285} C_VEL
LIN {X 0,Y 242.841,Z 787.214,A -85,B 0,C 180,E1 12346.505,E2 12346.505} C_VEL
LIN {X 0,Y 241.588,Z 790.508,A -85,B 0,C 180,E1 12341.943,E2 12341.943} C_VEL
LIN {X 0,Y 240.986,Z 792.337,A -85,B 0,C 180,E1 12337.39,E2 12337.39} C_VEL
LIN {X 0,Y 240.802,Z 792.754,A -85,B 0,C 180,E1 12332.856,E2 12332.856} C_VEL
LIN {X 0,Y 240.948,Z 791.774,A -85,B 0,C 180,E1 12328.336,E2 12328.336} C_VEL
LIN {X 0,Y 241.498,Z 789.392,A -85,B 0,C 180,E1 12323.82,E2 12323.82} C_VEL
LIN {X 0,Y 242.756,Z 785.28,A -85,B 0,C 180,E1 12319.079,E2 12319.079} C_VEL
LIN {X 0,Y 245.096,Z 779.117,A -85,B 0,C 180,E1 12314.138,E2 12314.138} C_VEL
LIN {X 0,Y 248.442,Z 771.356,A -85,B 0,C 180,E1 12309.504,E2 12309.504} C_VEL
LIN {X 0,Y 252.715,Z 762.101,A -85,B 0,C 180,E1 12305.204,E2 12305.204} C_VEL
LIN {X 0,Y 257.818,Z 751.319,A -85,B 0,C 180,E1 12301.221,E2 12301.221} C_VEL
LIN {X 0,Y 263.443,Z 739.334,A -85,B 0,C 180,E1 12297.646,E2 12297.646} C_VEL
LIN {X 0,Y 269.546,Z 725.855,A -85,B 0,C 180,E1 12294.382,E2 12294.382} C_VEL
LIN {X 0,Y 275.9,Z 710.909,A -85,B 0,C 180,E1 12291.44,E2 12291.44} C_VEL
LIN {X 0,Y 282.204,Z 694.774,A -85,B 0,C 180,E1 12288.864,E2 12288.864} C_VEL
LIN {X 0,Y 288.269,Z 677.465,A -85,B 0,C 180,E1 12286.625,E2 12286.625} C_VEL
LIN {X 0,Y 293.684,Z 659.78,A -85,B 0,C 180,E1 12284.777,E2 12284.777} C_VEL
LIN {X 0,Y 297.438,Z 645.78,A -85,B 0,C 180,E1 12283.575,E2 12283.575} C_VEL
LIN {X 0,Y 298.572,Z 638.859,A -85,B 0,C 180,E1 12282.926,E2 12282.926} C_VEL
LIN {X 0,Y 298.503,Z 620.733,A -85,B 0,C 180,E1 12280.807,E2 12280.807} C_VEL
LIN {X 0,Y 299.031,Z 614.574,A -85,B 0,C 180,E1 12280.351,E2 12280.351} C_VEL
LIN {X 0,Y 305.079,Z 578.179,A -85,B 0,C 180,E1 12278.766,E2 12278.766} C_VEL
LIN {X 0,Y 312.911,Z 528.878,A -85,B 0,C 180,E1 12277.104,E2 12277.104} C_VEL
LIN {X 0,Y 319.223,Z 480.392,A -85,B 0,C 180,E1 12275.735,E2 12275.735} C_VEL
LIN {X 0,Y 320.886,Z 464.637,A -85,B 0,C 180,E1 12275.322,E2 12275.322} C_VEL
LIN {X 0,Y 314.123,Z 477.665,A -85,B 0,C 180,E1 12273.961,E2 12273.961} C_VEL
LIN {X 0,Y 308.339,Z 486.885,A -85,B 0,C 180,E1 12272.596,E2 12272.596} C_VEL
LIN {X 0,Y 306.917,Z 489.484,A -85,B 0,C 180,E1 12272.268,E2 12272.268} C_VEL
LIN {X 0,Y 305.623,Z 492.85,A -85,B 0,C 180,E1 12272.047,E2 12272.047} C_VEL
LIN {X 0,Y 300.8,Z 506.514,A -85,B 0,C 180,E1 12271.307,E2 12271.307} C_VEL
LIN {X 0,Y 298.126,Z 513.085,A -85,B 0,C 180,E1 12270.815,E2 12270.815} C_VEL
LIN {X 0,Y 292.773,Z 530.323,A -85,B 0,C 180,E1 12270.237,E2 12270.237} C_VEL
LIN {X 0,Y 288.223,Z 542.321,A -85,B 0,C 180,E1 12269.532,E2 12269.532} C_VEL
LIN {X 0,Y 284.539,Z 550.459,A -85,B 0,C 180,E1 12268.807,E2 12268.807} C_VEL
LIN {X 0,Y 279.576,Z 564.612,A -85,B 0,C 180,E1 12268.228,E2 12268.228} C_VEL
LIN {X 0,Y 275.237,Z 574.739,A -85,B 0,C 180,E1 12267.476,E2 12267.476} C_VEL
LIN {X 0,Y 272.279,Z 580.707,A -85,B 0,C 180,E1 12266.807,E2 12266.807} C_VEL
LIN {X 0,Y 267.648,Z 592.797,A -85,B 0,C 180,E1 12266.227,E2 12266.227} C_VEL
LIN {X 0,Y 263.769,Z 600.971,A -85,B 0,C 180,E1 12265.454,E2 12265.454} C_VEL
LIN {X 0,Y 261.12,Z 605.717,A -85,B 0,C 180,E1 12264.751,E2 12264.751} C_VEL
LIN {X 0,Y 257.052,Z 615.47,A -85,B 0,C 180,E1 12264.183,E2 12264.183} C_VEL
LIN {X 0,Y 253.823,Z 621.84,A -85,B 0,C 180,E1 12263.445,E2 12263.445} C_VEL
LIN {X 0,Y 251.318,Z 625.627,A -85,B 0,C 180,E1 12262.63,E2 12262.63} C_VEL
LIN {X 0,Y 247.782,Z 633.73,A -85,B 0,C 180,E1 12262.042,E2 12262.042} C_VEL
LIN {X 0,Y 244.928,Z 638.734,A -85,B 0,C 180,E1 12261.305,E2 12261.305} C_VEL
LIN {X 0,Y 243.395,Z 640.812,A -85,B 0,C 180,E1 12260.689,E2 12260.689} C_VEL
LIN {X 0,Y 242.637,Z 641.319,A -85,B 0,C 180,E1 12260.174,E2 12260.174} C_VEL
LIN {X 0,Y 241.634,Z 658.246,A -85,B 0,C 180,E1 12258.705,E2 12258.705} C_VEL
LIN {X 0,Y 240.41,Z 674.881,A -85,B 0,C 180,E1 12256.802,E2 12256.802} C_VEL
LIN {X 0,Y 239.095,Z 690.405,A -85,B 0,C 180,E1 12254.532,E2 12254.532} C_VEL
LIN {X 0,Y 237.757,Z 705.408,A -85,B 0,C 180,E1 12251.77,E2 12251.77} C_VEL
LIN {X 0,Y 236.616,Z 719.158,A -85,B 0,C 180,E1 12248.579,E2 12248.579} C_VEL
LIN {X 0,Y 235.881,Z 730.212,A -85,B 0,C 180,E1 12245.352,E2 12245.352} C_VEL
LIN {X 0,Y 235.523,Z 738.838,A -85,B 0,C 180,E1 12242.191,E2 12242.191} C_VEL
LIN {X 0,Y 235.564,Z 746.66,A -85,B 0,C 180,E1 12238.542,E2 12238.542} C_VEL
LIN {X 0,Y 236.084,Z 752.354,A -85,B 0,C 180,E1 12234.898,E2 12234.898} C_VEL
LIN {X 0,Y 237.128,Z 756.192,A -85,B 0,C 180,E1 12231.27,E2 12231.27} C_VEL
LIN {X 0,Y 238.755,Z 758.227,A -85,B 0,C 180,E1 12227.669,E2 12227.669} C_VEL
LIN {X 0,Y 241.005,Z 758.435,A -85,B 0,C 180,E1 12224.109,E2 12224.109} C_VEL
LIN {X 0,Y 244.132,Z 756.711,A -85,B 0,C 180,E1 12220.377,E2 12220.377} C_VEL
LIN {X 0,Y 248.02,Z 752.818,A -85,B 0,C 180,E1 12216.73,E2 12216.73} C_VEL
LIN {X 0,Y 252.044,Z 747.543,A -85,B 0,C 180,E1 12213.622,E2 12213.622} C_VEL
LIN {X 0,Y 256.659,Z 740.406,A -85,B 0,C 180,E1 12210.604,E2 12210.604} C_VEL
LIN {X 0,Y 261.814,Z 731.044,A -85,B 0,C 180,E1 12207.68,E2 12207.68} C_VEL
LIN {X 0,Y 267.105,Z 720.092,A -85,B 0,C 180,E1 12205.06,E2 12205.06} C_VEL
LIN {X 0,Y 270.55,Z 712.502,A -85,B 0,C 180,E1 12203.554,E2 12203.554} C_VEL
LIN {X 0,Y 274.181,Z 711.227,A -85,B 0,C 180,E1 12203.009,E2 12203.009} C_VEL
LIN {X 0,Y 277.94,Z 709.315,A -85,B 0,C 180,E1 12202.559,E2 12202.559} C_VEL
LIN {X 0,Y 282.377,Z 707.212,A -85,B 0,C 180,E1 12202.033,E2 12202.033} C_VEL
LIN {X 0,Y 275.989,Z 725.231,A -85,B 0,C 180,E1 12199.846,E2 12199.846} C_VEL
LIN {X 0,Y 269.356,Z 742.116,A -85,B 0,C 180,E1 12197.306,E2 12197.306} C_VEL
LIN {X 0,Y 262.737,Z 757.582,A -85,B 0,C 180,E1 12194.445,E2 12194.445} C_VEL
LIN {X 0,Y 255.928,Z 772.459,A -85,B 0,C 180,E1 12191.022,E2 12191.022} C_VEL
LIN {X 0,Y 249.496,Z 786.216,A -85,B 0,C 180,E1 12187.11,E2 12187.11} C_VEL
LIN {X 0,Y 244.079,Z 797.768,A -85,B 0,C 180,E1 12183.013,E2 12183.013} C_VEL
LIN {X 0,Y 239.187,Z 808.797,A -85,B 0,C 180,E1 12178.113,E2 12178.113} C_VEL
LIN {X 0,Y 235.808,Z 817.431,A -85,B 0,C 180,E1 12173.224,E2 12173.224} C_VEL
LIN {X 0,Y 233.587,Z 824.584,A -85,B 0,C 180,E1 12167.95,E2 12167.95} C_VEL
LIN {X 0,Y 232.616,Z 829.663,A -85,B 0,C 180,E1 12162.915,E2 12162.915} C_VEL
LIN {X 0,Y 232.448,Z 832.963,A -85,B 0,C 180,E1 12158.161,E2 12158.161} C_VEL
LIN {X 0,Y 232.594,Z 834.771,A -85,B 0,C 180,E1 12153.697,E2 12153.697} C_VEL
LIN {X 0,Y 232.666,Z 835.319,A -85,B 0,C 180,E1 12149.507,E2 12149.507} C_VEL
LIN {X 0,Y 232.527,Z 834.688,A -85,B 0,C 180,E1 12145.066,E2 12145.066} C_VEL
LIN {X 0,Y 232.406,Z 832.687,A -85,B 0,C 180,E1 12140.341,E2 12140.341} C_VEL
LIN {X 0,Y 232.81,Z 829.043,A -85,B 0,C 180,E1 12135.322,E2 12135.322} C_VEL
LIN {X 0,Y 234.364,Z 823.22,A -85,B 0,C 180,E1 12129.783,E2 12129.783} C_VEL
LIN {X 0,Y 237.066,Z 816.178,A -85,B 0,C 180,E1 12124.787,E2 12124.787} C_VEL
LIN {X 0,Y 241.377,Z 806.723,A -85,B 0,C 180,E1 12119.644,E2 12119.644} C_VEL
LIN {X 0,Y 246.954,Z 795.635,A -85,B 0,C 180,E1 12114.905,E2 12114.905} C_VEL
LIN {X 0,Y 253.564,Z 782.789,A -85,B 0,C 180,E1 12110.59,E2 12110.59} C_VEL
LIN {X 0,Y 260.557,Z 769.133,A -85,B 0,C 180,E1 12106.916,E2 12106.916} C_VEL
LIN {X 0,Y 267.978,Z 753.872,A -85,B 0,C 180,E1 12103.627,E2 12103.627} C_VEL
LIN {X 0,Y 275.358,Z 737.614,A -85,B 0,C 180,E1 12100.813,E2 12100.813} C_VEL
LIN {X 0,Y 282.277,Z 720.914,A -85,B 0,C 180,E1 12098.481,E2 12098.481} C_VEL
LIN {X 0,Y 288.968,Z 702.643,A -85,B 0,C 180,E1 12096.44,E2 12096.44} C_VEL
LIN {X 0,Y 295.361,Z 682.417,A -85,B 0,C 180,E1 12094.653,E2 12094.653} C_VEL
LIN {X 0,Y 302.918,Z 655.825,A -85,B 0,C 180,E1 12092.773,E2 12092.773} C_VEL
LIN {X 0,Y 310.018,Z 628.339,A -85,B 0,C 180,E1 12091.276,E2 12091.276} C_VEL
LIN {X 0,Y 311.036,Z 624.07,A -85,B 0,C 180,E1 12091.071,E2 12091.071} C_VEL
LIN {X 0,Y 305.414,Z 634.141,A -85,B 0,C 180,E1 12090.71,E2 12090.71} C_VEL
LIN {X 0,Y 300.579,Z 641.387,A -85,B 0,C 180,E1 12090.272,E2 12090.272} C_VEL
LIN {X 0,Y 294.884,Z 650.756,A -85,B 0,C 180,E1 12089.896,E2 12089.896} C_VEL
LIN {X 0,Y 290.075,Z 657.284,A -85,B 0,C 180,E1 12089.41,E2 12089.41} C_VEL
LIN {X 0,Y 285.257,Z 664.383,A -85,B 0,C 180,E1 12089.042,E2 12089.042} C_VEL
LIN {X 0,Y 281.18,Z 669.304,A -85,B 0,C 180,E1 12088.559,E2 12088.559} C_VEL
LIN {X 0,Y 276.714,Z 675.329,A -85,B 0,C 180,E1 12088.156,E2 12088.156} C_VEL
LIN {X 0,Y 272.507,Z 679.789,A -85,B 0,C 180,E1 12087.535,E2 12087.535} C_VEL
LIN {X 0,Y 268.236,Z 684.881,A -85,B 0,C 180,E1 12087.049,E2 12087.049} C_VEL
LIN {X 0,Y 264.988,Z 687.768,A -85,B 0,C 180,E1 12086.438,E2 12086.438} C_VEL
LIN {X 0,Y 262.387,Z 700.841,A -85,B 0,C 180,E1 12084.902,E2 12084.902} C_VEL
LIN {X 0,Y 259.363,Z 713.232,A -85,B 0,C 180,E1 12083.034,E2 12083.034} C_VEL
LIN {X 0,Y 255.925,Z 724.497,A -85,B 0,C 180,E1 12080.825,E2 12080.825} C_VEL
LIN {X 0,Y 252.567,Z 733.844,A -85,B 0,C 180,E1 12078.463,E2 12078.463} C_VEL
LIN {X 0,Y 248.914,Z 742.297,A -85,B 0,C 180,E1 12075.612,E2 12075.612} C_VEL
LIN {X 0,Y 245.672,Z 748.539,A -85,B 0,C 180,E1 12072.695,E2 12072.695} C_VEL
LIN {X 0,Y 242.665,Z 753.122,A -85,B 0,C 180,E1 12069.486,E2 12069.486} C_VEL
LIN {X 0,Y 240.188,Z 755.695,A -85,B 0,C 180,E1 12066.213,E2 12066.213} C_VEL
LIN {X 0,Y 238.26,Z 756.417,A -85,B 0,C 180,E1 12062.886,E2 12062.886} C_VEL
LIN {X 0,Y 236.87,Z 755.312,A -85,B 0,C 180,E1 12059.515,E2 12059.515} C_VEL
LIN {X 0,Y 235.973,Z 752.333,A -85,B 0,C 180,E1 12056.112,E2 12056.112} C_VEL
LIN {X 0,Y 235.551,Z 747.39,A -85,B 0,C 180,E1 12052.683,E2 12052.683} C_VEL
LIN {X 0,Y 235.557,Z 740.871,A -85,B 0,C 180,E1 12049.483,E2 12049.483} C_VEL
LIN {X 0,Y 235.907,Z 732.95,A -85,B 0,C 180,E1 12046.519,E2 12046.519} C_VEL
LIN {X 0,Y 236.578,Z 722.976,A -85,B 0,C 180,E1 12043.615,E2 12043.615} C_VEL
LIN {X 0,Y 237.477,Z 711.358,A -85,B 0,C 180,E1 12040.955,E2 12040.955} C_VEL
LIN {X 0,Y 238.487,Z 698.348,A -85,B 0,C 180,E1 12038.607,E2 12038.607} C_VEL
LIN {X 0,Y 238.855,Z 693.829,A -85,B 0,C 180,E1 12037.867,E2 12037.867} C_VEL
LIN {X 0,Y 239.832,Z 693.832,A -85,B 0,C 180,E1 12037.187,E2 12037.187} C_VEL
LIN {X 0,Y 242,Z 692.542,A -85,B 0,C 180,E1 12036.373,E2 12036.373} C_VEL
LIN {X 0,Y 244.845,Z 690.235,A -85,B 0,C 180,E1 12035.64,E2 12035.64} C_VEL
LIN {X 0,Y 247.529,Z 688.817,A -85,B 0,C 180,E1 12034.647,E2 12034.647} C_VEL
LIN {X 0,Y 251.071,Z 686.009,A -85,B 0,C 180,E1 12033.765,E2 12033.765} C_VEL
LIN {X 0,Y 252.526,Z 684.847,A -85,B 0,C 180,E1 12033.421,E2 12033.421} C_VEL
LIN {X 0,Y 256.455,Z 682.184,A -85,B 0,C 180,E1 12032.357,E2 12032.357} C_VEL
LIN {X 0,Y 262.133,Z 677.216,A -85,B 0,C 180,E1 12031.274,E2 12031.274} C_VEL
LIN {X 0,Y 267.316,Z 672.989,A -85,B 0,C 180,E1 12030.201,E2 12030.201} C_VEL
LIN {X 0,Y 273.823,Z 666.352,A -85,B 0,C 180,E1 12029.255,E2 12029.255} C_VEL
LIN {X 0,Y 279.583,Z 660.69,A -85,B 0,C 180,E1 12028.338,E2 12028.338} C_VEL
LIN {X 0,Y 285.491,Z 653.369,A -85,B 0,C 180,E1 12027.717,E2 12027.717} C_VEL
LIN {X 0,Y 287.629,Z 650.444,A -85,B 0,C 180,E1 12027.514,E2 12027.514} C_VEL
LIN {X 0,Y 293.707,Z 643.104,A -85,B 0,C 180,E1 12026.763,E2 12026.763} C_VEL
LIN {X 0,Y 299.724,Z 633.727,A -85,B 0,C 180,E1 12026.259,E2 12026.259} C_VEL
LIN {X 0,Y 301.359,Z 631.025,A -85,B 0,C 180,E1 12026.123,E2 12026.123} C_VEL
LIN {X 0,Y 303.476,Z 628.196,A -85,B 0,C 180,E1 12025.848,E2 12025.848} C_VEL
LIN {X 0,Y 298.857,Z 647.267,A -85,B 0,C 180,E1 12024.554,E2 12024.554} C_VEL
LIN {X 0,Y 293.22,Z 666.131,A -85,B 0,C 180,E1 12022.933,E2 12022.933} C_VEL
LIN {X 0,Y 286.761,Z 684.438,A -85,B 0,C 180,E1 12020.947,E2 12020.947} C_VEL
LIN {X 0,Y 279.786,Z 701.591,A -85,B 0,C 180,E1 12018.613,E2 12018.613} C_VEL
LIN {X 0,Y 272.64,Z 717.322,A -85,B 0,C 180,E1 12015.956,E2 12015.956} C_VEL
LIN {X 0,Y 265.554,Z 731.64,A -85,B 0,C 180,E1 12012.961,E2 12012.961} C_VEL
LIN {X 0,Y 258.321,Z 745.279,A -85,B 0,C 180,E1 12009.404,E2 12009.404} C_VEL
LIN {X 0,Y 251.652,Z 757.303,A -85,B 0,C 180,E1 12005.457,E2 12005.457} C_VEL
LIN {X 0,Y 246.042,Z 767.228,A -85,B 0,C 180,E1 12001.344,E2 12001.344} C_VEL
LIN {X 0,Y 241.295,Z 775.736,A -85,B 0,C 180,E1 11996.851,E2 11996.851} C_VEL
LIN {X 0,Y 237.58,Z 782.735,A -85,B 0,C 180,E1 11991.997,E2 11991.997} C_VEL
LIN {X 0,Y 235.085,Z 787.898,A -85,B 0,C 180,E1 11987.066,E2 11987.066} C_VEL
LIN {X 0,Y 233.658,Z 791.342,A -85,B 0,C 180,E1 11982.104,E2 11982.104} C_VEL
LIN {X 0,Y 233.021,Z 793.101,A -85,B 0,C 180,E1 11977.396,E2 11977.396} C_VEL
LIN {X 0,Y 232.832,Z 793.453,A -85,B 0,C 180,E1 11972.708,E2 11972.708} C_VEL
LIN {X 0,Y 233,Z 792.414,A -85,B 0,C 180,E1 11968.033,E2 11968.033} C_VEL
LIN {X 0,Y 233.62,Z 789.977,A -85,B 0,C 180,E1 11963.364,E2 11963.364} C_VEL
LIN {X 0,Y 235.012,Z 785.82,A -85,B 0,C 180,E1 11958.465,E2 11958.465} C_VEL
LIN {X 0,Y 237.415,Z 779.945,A -85,B 0,C 180,E1 11953.61,E2 11953.61} C_VEL
LIN {X 0,Y 240.966,Z 772.219,A -85,B 0,C 180,E1 11948.839,E2 11948.839} C_VEL
LIN {X 0,Y 245.481,Z 763.003,A -85,B 0,C 180,E1 11944.422,E2 11944.422} C_VEL
LIN {X 0,Y 250.881,Z 752.213,A -85,B 0,C 180,E1 11940.323,E2 11940.323} C_VEL
LIN {X 0,Y 256.749,Z 740.332,A -85,B 0,C 180,E1 11936.695,E2 11936.695} C_VEL
LIN {X 0,Y 263.122,Z 726.899,A -85,B 0,C 180,E1 11933.373,E2 11933.373} C_VEL
LIN {X 0,Y 269.416,Z 712.797,A -85,B 0,C 180,E1 11930.529,E2 11930.529} C_VEL
LIN {X 0,Y 275.588,Z 697.816,A -85,B 0,C 180,E1 11928.054,E2 11928.054} C_VEL
LIN {X 0,Y 281.891,Z 680.803,A -85,B 0,C 180,E1 11925.767,E2 11925.767} C_VEL
LIN {X 0,Y 287.65,Z 663.022,A -85,B 0,C 180,E1 11923.841,E2 11923.841} C_VEL
LIN {X 0,Y 292.886,Z 643.95,A -85,B 0,C 180,E1 11922.2,E2 11922.2} C_VEL
LIN {X 0,Y 297.23,Z 624.353,A -85,B 0,C 180,E1 11920.883,E2 11920.883} C_VEL
LIN {X 0,Y 299.031,Z 614.574,A -85,B 0,C 180,E1 11920.351,E2 11920.351} C_VEL
LIN {X 0,Y 299.693,Z 607.327,A -85,B 0,C 180,E1 11919.829,E2 11919.829} C_VEL
LIN {X 0,Y 299.264,Z 589.375,A -85,B 0,C 180,E1 11918.098,E2 11918.098} C_VEL
LIN {X 0,Y 299.981,Z 582.036,A -85,B 0,C 180,E1 11917.649,E2 11917.649} C_VEL
LIN {X 0,Y 308.029,Z 533.513,A -85,B 0,C 180,E1 11915.985,E2 11915.985} C_VEL
LIN {X 0,Y 314.539,Z 485.827,A -85,B 0,C 180,E1 11914.615,E2 11914.615} C_VEL
LIN {X 0,Y 309.177,Z 494.119,A -85,B 0,C 180,E1 11913.408,E2 11913.408} C_VEL
LIN {X 0,Y 303.559,Z 509.695,A -85,B 0,C 180,E1 11912.599,E2 11912.599} C_VEL
LIN {X 0,Y 300.893,Z 516.173,A -85,B 0,C 180,E1 11912.149,E2 11912.149} C_VEL
LIN {X 0,Y 295.38,Z 533.351,A -85,B 0,C 180,E1 11911.59,E2 11911.59} C_VEL
LIN {X 0,Y 290.547,Z 545.71,A -85,B 0,C 180,E1 11910.891,E2 11910.891} C_VEL
LIN {X 0,Y 286.846,Z 553.893,A -85,B 0,C 180,E1 11910.217,E2 11910.217} C_VEL
LIN {X 0,Y 281.664,Z 568.154,A -85,B 0,C 180,E1 11909.638,E2 11909.638} C_VEL
LIN {X 0,Y 277.004,Z 578.722,A -85,B 0,C 180,E1 11908.868,E2 11908.868} C_VEL
LIN {X 0,Y 274.139,Z 584.31,A -85,B 0,C 180,E1 11908.296,E2 11908.296} C_VEL
LIN {X 0,Y 269.329,Z 596.431,A -85,B 0,C 180,E1 11907.71,E2 11907.71} C_VEL
LIN {X 0,Y 265.023,Z 605.279,A -85,B 0,C 180,E1 11906.889,E2 11906.889} C_VEL
